// ---- WIND TURBINE/FB_WatsAppResponse.TcPOU
FUNCTION_BLOCK FB_WatsAppResponse
VAR_INPUT
	bSend             : BOOL;
END_VAR
VAR_OUTPUT
	wind_speed		  : Lreal;
	bBusy             : BOOL;
    bError            : BOOL;
END_VAR
VAR
	fbRequest         : FB_IotHttpRequest;
    fbJson            : FB_JsonDomParser;
    nState            : UDINT;
    RisingEdge        : R_TRIG;

    bGetContentResult : BOOL;
    sContent          : STRING(511);

    bGetJsonResult    : BOOL;
    jsonDoc           : SJsonValue;
    jsonVal           : SJsonValue;
	jsonWind           : SJsonValue;

    nReqCount         : UDINT;
    nResCount         : UDINT;
    nValidResCount    : UDINT;
    nErrCount         : UDINT;
	bHasMember		  : BOOL;
	bHasMember2		  : BOOL;
END_VAR
VAR_IN_OUT
	 fbClient          : FB_IotHttpClient;
END_VAR

RisingEdge(CLK:= bSend);
CASE nState OF
0:
    IF RisingEdge.Q THEN
        IF fbRequest.SendRequest(sUri:= '/cebc385e-7c19-40b8-aaac-81ec04618ab7',
                                 fbClient:= fbClient, 
                                 eRequestType:= ETcIotHttpRequestType.HTTP_POST, 0, 0, 0) THEN
            nState:= 1;
            nReqCount:= nReqCount+1;
            bBusy:= TRUE;
            bError:= FALSE;
        END_IF
    END_IF
1:
    IF NOT fbRequest.bBusy THEN
        bError:= TRUE;
        IF NOT fbRequest.bError THEN
            bGetContentResult:= fbRequest.GetContent(pContent:= ADR(sContent), 
                                                     nContentSize:= SIZEOF(sContent), 
                                                     bSetNullTermination:= TRUE);
            IF fbRequest.nStatusCode >= 200 AND fbRequest.nStatusCode < 300 THEN
                bGetJsonResult:= FALSE;
                jsonDoc:= fbRequest.GetJsonDomContent(fbJson);
//                IF jsonDoc <> 0 THEN
//                    bHasMember := fbJson.HasMember(jsonDoc, 'current');
//					IF (bHasMember) THEN
//						bHasMember := FALSE;
//						jsonVal := fbJson.FindMember(jsonDoc, 'current');
//					END_IF
					
//					bHasMember2 := fbJson.HasMember(jsonVal, 'wind_mph');
//					IF (bHasMember2) THEN
//						bHasMember2 := FALSE;
//						jsonWind := fbJson.FindMember(jsonVal, 'wind_mph');
//						wind_speed := fbJson.GetDouble(jsonWind);
//						WindSpeed := fbJson.GetDouble(jsonWind);
//					END_IF
					
//                    nValidResCount:= nValidResCount+1;
//                    bError:= FALSE;
//                END_IF
                nResCount:= nResCount+1;
            END_IF
        END_IF
        nState:= 0;
        bBusy:= FALSE;
        IF bError THEN
            nErrCount:= nErrCount+1;
        END_IF
    END_IF
END_CASE

END_FUNCTION_BLOCK

// ---- BLINDS/BackgroundComms.TcPOU
PROGRAM BackgroundComms
VAR

	HubTXBuffer								:		ARRAY [0..2] OF ComBuffer;
	HubRXBuffer								:		ARRAY [0..2] OF ComBuffer;
                                			        
	HubCommIn AT %I*						:		ARRAY [0..2] OF KL6inData22B;
	HubCommOut AT %Q*						:		ARRAY [0..2] OF KL6outData22B;
                                			        
	HubSerialLineControl					:		ARRAY [0..2] OF SerialLineControl;
                                			        
	i										:		INT;
                                			
	BlindCommandTable 						:		ARRAY [0..2] OF StructBlindControl := [(JogTimeInt:=3000)];
	                            			
	OfficeBlindSellection					:		ARRAY [0..2] OF BOOL;
	                            			
	KitchenBlindSelection					:		BOOL;
	                            			
	BoardroomBlindSellection				:		ARRAY [0..1] OF BOOL;
                                			
	StaffRoomTempDownButton					:		BOOL;
	StaffRoomTempUpButton					:		BOOL;
	StaffRoomTempDownButtonFlag				:		BOOL;
	StaffRoomTempUpButtonFlag				:		BOOL;
	ResetFlagTime 							: 		TON;
                                			
	BlindSelection							:		Selection;
                                			
	UseStaffRoomVisu 						: 		BOOL;
                                			
	Up										:		BOOL;
	Down									:		BOOL;
                                			
	rtBlindsBoardRoomUp						:		R_TRIG;
	rtBlindsBoardRoomDown					:		R_TRIG;
	rtBlindsBoardRoomStop					:		R_TRIG;
	                            			
	rtBlindsOfficeUp						:		R_TRIG;

	(*Office Blinds Triggers *)
	rtBlindsOfficeAreaWall1_3				:		R_TRIG;
	rtBlindsOfficeAreaWall1_3_10_13			:		R_TRIG;
	rtBlindsOfficeAreaWall1_9				:		R_TRIG;
	rtBlindsOfficeAreaWall4_9				:		R_TRIG;
	rtBlindsOfficeAreaWall4_13				:		R_TRIG;
	rtBlindsOfficeAreaWall10_13				:		R_TRIG;
	rtBlindsOfficeAreaWallAll				:		R_TRIG;
	rtBlindsOfficeAreaWallAllFalse			:		R_TRIG;
	
	(*Kitchen Blinds Triggers *)
	rtBlindsKitchenAreaWallAll				:		R_TRIG;
	rtBlindsKitchenAreaWallAllFalse				:		R_TRIG;
	
	(*Boardroom Blinds Triggers *)
	rtBlindsBoardroomAreaWall1_7			:		R_TRIG;
	rtBlindsBoardroomAreaWall8_16			:		R_TRIG;
	rtBlindsBoardroomAreaWallAll			:		R_TRIG;
	rtBlindsBoardroomAreaWallAllFalse		:		R_TRIG;
	
	rtBlindsOfficeAreaWallStop				:		R_TRIG;


	xBlindsOfficeAreaWall1_3Flag			:		BOOL;
	xBlindsOfficeAreaWall4_9Flag			:		BOOL;
	xBlindsOfficeAreaWall10_13Flag			:		BOOL;

	rtBlindsBoardRoomCP67Up					:		R_TRIG;
	rtBlindsBoardRoomCP67Down				:		R_TRIG;
	rtBlindsBoardRoomCP67Stop				:		R_TRIG;


	rtBoardRoom_PrivacyMode					:		R_TRIG;
	rtBoardRoom_SceneryMode					:		R_TRIG;
	rtBoardRoom_ProjectorMode				:		R_TRIG;
	rtBoardRoom_MeetingMode					:		R_TRIG;
                                    		        
	rtDeskArea_PrivacyMode					:		R_TRIG;
	rtDeskArea_SceneryMode					:		R_TRIG;
	rtDeskArea_NightMode					:		R_TRIG;
	rtDeskArea_MorningMode					:		R_TRIG;
                                        	        
	rtKitchenArea_PrivacyMode				:		R_TRIG;
	rtKitchenArea_SceneryMode				:		R_TRIG;
	rtKitchenArea_NightMode					:		R_TRIG;
	rtKitchenArea_MorningMode				:		R_TRIG;
                                        	        
	rtEntireBuilding_CleaningMode			:		R_TRIG;


END_VAR


VAR CONSTANT

	HubCount								:		INT := 2; (* Hub count starts at 0, setting 2 = 3 hubs *)

END_VAR

(* Serial line control for Office Area *)
HubSerialLineControl[0](
	Mode:= SERIALLINEMODE_KL6_22B_STANDARD ,
	pComIn:= ADR( HubCommIn[0]),
	pComOut:= ADR( HubCommOut[0]),
	SizeComIn:=  SIZEOF(HubCommIn[0]),
	TxBuffer:= HubTXBuffer[0] ,
	RxBuffer:= HubRXBuffer[0] ,
	Error=> ,
	ErrorID=> );

(* Serial line control for Boardroom *)
HubSerialLineControl[1](
	Mode:= SERIALLINEMODE_KL6_22B_STANDARD ,
	pComIn:= ADR( HubCommIn[1]),
	pComOut:= ADR( HubCommOut[1]),
	SizeComIn:=  SIZEOF(HubCommIn[1]),
	TxBuffer:= HubTXBuffer[1] ,
	RxBuffer:= HubRXBuffer[1] ,
	Error=> ,
	ErrorID=> );

(*Serial line control for reception *)
HubSerialLineControl[2](
	Mode:= SERIALLINEMODE_KL6_22B_STANDARD ,
	pComIn:= ADR( HubCommIn[2]),
	pComOut:= ADR( HubCommOut[2]),
	SizeComIn:=  SIZEOF(HubCommIn[2]),
	TxBuffer:= HubTXBuffer[2] ,
	RxBuffer:= HubRXBuffer[2] ,
	Error=> ,
	ErrorID=> );

(* Check trigger for boardRoom blinds*)
rtBlindsBoardRoomDown(CLK:= PassADSBlindInfo[2].0 , Q=> );
IF rtBlindsBoardRoomDown.Q THEN
	SetBoardroomAreaBlindsAll();
	BlindCommandTable[1].xCommandDown := TRUE;
END_IF

rtBlindsBoardRoomUp(CLK:= PassADSBlindInfo[3].0 , Q=> );
IF rtBlindsBoardRoomUp.Q THEN
	SetBoardroomAreaBlindsAll();
	BlindCommandTable[1].xCommandUp := TRUE;
END_IF

(*Desk Area Blinds selection******************************************************************)
(*Select Office Blinds and combitanions*)

rtBlindsOfficeAreaWall1_3(CLK := OfficeBlindSellection[0] AND (NOT OfficeBlindSellection[1]) AND (NOT OfficeBlindSellection[2]));
rtBlindsOfficeAreaWall1_3_10_13(CLK := OfficeBlindSellection[0] AND (NOT OfficeBlindSellection[1]) AND OfficeBlindSellection[2]);
rtBlindsOfficeAreaWall1_9(CLK := OfficeBlindSellection[0] AND OfficeBlindSellection[1] AND (NOT OfficeBlindSellection[2]));
rtBlindsOfficeAreaWallAll(CLK := OfficeBlindSellection[0] AND OfficeBlindSellection[1] AND OfficeBlindSellection[2]);
rtBlindsOfficeAreaWall4_9(CLK := (NOT OfficeBlindSellection[0]) AND OfficeBlindSellection[1] AND (NOT OfficeBlindSellection[2]));
rtBlindsOfficeAreaWall4_13(CLK := (NOT OfficeBlindSellection[0]) AND OfficeBlindSellection[1] AND OfficeBlindSellection[2]);
rtBlindsOfficeAreaWall10_13(CLK := (NOT OfficeBlindSellection[0]) AND (NOT OfficeBlindSellection[1]) AND OfficeBlindSellection[2]);
rtBlindsOfficeAreaWallAllFalse(CLK := (NOT OfficeBlindSellection[0]) AND (NOT OfficeBlindSellection[1]) AND (NOT OfficeBlindSellection[2]));

IF rtBlindsOfficeAreaWall1_3.Q THEN
	SetOfficeAreaBlinds1_3();
END_IF

IF rtBlindsOfficeAreaWall1_3_10_13.Q THEN
	SetOfficeAreaBlinds1_3_10_13();
END_IF

IF rtBlindsOfficeAreaWall1_9.Q THEN
	SetOfficeAreaBlinds1_9();
END_IF

IF rtBlindsOfficeAreaWallAll.Q THEN
	SetOfficeAreaBlindsAll();
END_IF

IF rtBlindsOfficeAreaWall4_9.Q THEN
	SetOfficeAreaBlinds4_9();
END_IF

IF rtBlindsOfficeAreaWall4_13.Q THEN
	SetOfficeAreaBlinds4_13();
END_IF

IF rtBlindsOfficeAreaWall10_13.Q THEN
	SetOfficeAreaBlinds10_13();
END_IF

IF rtBlindsOfficeAreaWallAllFalse.Q THEN
	SetOfficeAreaBlindsAllFalse();
END_IF


(*Kitchen Area Blinds selection******************************************************************)
(*Select Kitchen Blinds for Lond Wall*)

rtBlindsKitchenAreaWallAll(CLK := KitchenBlindSelection);
rtBlindsKitchenAreaWallAllFalse(CLK := NOT KitchenBlindSelection);

IF rtBlindsKitchenAreaWallAll.Q THEN
	SetKitchenAreaBlindsAll();
END_IF

IF rtBlindsKitchenAreaWallAllFalse.Q THEN
	SetKitchenAreaBlindsAllFalse();
END_IF

(*Boardroom Area Blinds selection******************************************************************)
(*Select Boardroom Blinds for Lond Wall*)

rtBlindsBoardroomAreaWall1_7(CLK := BoardroomBlindSellection[1] AND (NOT BoardroomBlindSellection[0]));		
rtBlindsBoardroomAreaWall8_16(CLK := (NOT BoardroomBlindSellection[1]) AND BoardroomBlindSellection[0]);
rtBlindsBoardroomAreaWallAll(CLK := BoardroomBlindSellection[0] AND BoardroomBlindSellection[1]);
rtBlindsBoardroomAreaWallAllFalse(CLK := (NOT BoardroomBlindSellection[0]) AND (NOT BoardroomBlindSellection[1]));

IF rtBlindsBoardroomAreaWall1_7.Q THEN
	SetBoardRoomBlinds1_7();
END_IF

IF rtBlindsBoardroomAreaWall8_16.Q THEN
	SetBoardRoomBlinds8_16();
END_IF

IF rtBlindsBoardroomAreaWallAll.Q THEN
	SetBoardroomAreaBlindsAll();
END_IF

IF rtBlindsBoardroomAreaWallAllFalse.Q THEN
	SetBoardroomAreaBlindsAllFalse();
END_IF

(*Boardroom Blind Modes**************************************************************************)
                                                                                        	
(*Board Room Privacy Mode *)                                                            	
rtBoardRoom_PrivacyMode(CLK:= BoardRoom_PrivacyMode , Q=> );                            	
IF rtBoardRoom_PrivacyMode.Q THEN                                                       	
	SetBoardRoomBlinds1_7();                                                            	
	BlindCommandTable[1].xCommandDown := TRUE;                                          	
	BoardRoom_PrivacyMode	:= FALSE;                                                   	
END_IF                                                                                  	
                                                                                        	
(*Board Room Scenery Mode *)                                                            	
rtBoardRoom_SceneryMode(CLK:= BoardRoom_SceneryMode , Q=> );                            	
IF rtBoardRoom_SceneryMode.Q THEN                                                       	
	SetBoardRoomBlinds8_16();                                                           	
	BlindCommandTable[1].xCommandUp := TRUE;                                            	
	BoardRoom_SceneryMode	:= FALSE;                                                   	
END_IF                                                                                  	
                                                                                        	
(*Board Room Projector Mode *)                                                          	
rtBoardRoom_ProjectorMode(CLK:= BoardRoom_ProjectorMode , Q=> );                        	
IF rtBoardRoom_ProjectorMode.Q THEN                                                     	
	SetBoardroomAreaBlindsAll();                                                        	
	BlindCommandTable[1].xCommandDown := TRUE;                                          	
	BoardRoom_ProjectorMode	:= FALSE;                                                   	
END_IF                                                                                  	
                                                                                        	
(*Meeting Room Mode *)                                                                 	
rtBoardRoom_ProjectorMode(CLK:= BoardRoom_ProjectorMode , Q=> );                        	
IF rtBoardRoom_ProjectorMode.Q THEN                                                     	
	SetBoardRoomBlinds1_7();                                                            	
	BlindCommandTable[1].xCommandDown := TRUE;                                          	
	BoardRoom_ProjectorMode	:= FALSE;                                                   	
END_IF                                                                                  	
                                                                                        	
                                                                                        	
(*Desk Area Blind Modes*****************************************************************	******)
                                                                                        	
(* Desk Area Privacy Mode*)                                                             	
rtDeskArea_PrivacyMode(CLK:= DeskArea_PrivacyMode OR PassADSBlindInfo[8].0  , Q=> );    	
IF rtDeskArea_PrivacyMode.Q THEN                                                        	
	SetOfficeAreaBlinds10_13();                                                         	
	BlindCommandTable[0].xCommandDown := TRUE;                                          	
	DeskArea_PrivacyMode	:= FALSE;                                                   	
END_IF                                                                                  	
                                                                                        	
(* Desk Area Scenery Mode*)                                                             	
rtDeskArea_SceneryMode(CLK:= DeskArea_SceneryMode OR  PassADSBlindInfo[11].0  , Q=> );  	
IF rtDeskArea_SceneryMode.Q THEN                                                        	
	SetOfficeAreaBlinds4_9();                                                           	
	BlindCommandTable[0].xCommandUp := TRUE;                                            	
	DeskArea_SceneryMode	:= FALSE;                                                   	
END_IF                                                                                  	
                                                                                        	
(* Desk Area Night Mode*)                                                               	
rtDeskArea_NightMode(CLK:= DeskArea_NightMode OR  PassADSBlindInfo[9].0 , Q=> );        	
IF rtDeskArea_NightMode.Q THEN                                                          	
	SetOfficeAreaBlinds1_9();                                                           	
	BlindCommandTable[0].xCommandDown := TRUE;                                          	
	DeskArea_NightMode	:= FALSE;                                                       	
END_IF                                                                                  	
                                                                                        	
(* Desk Area Morning Mode*)                                                             	
rtDeskArea_MorningMode(CLK:= DeskArea_MorningMode OR  PassADSBlindInfo[10].0 , Q=> );   	
IF rtDeskArea_MorningMode.Q THEN                                                        	
	SetOfficeAreaBlinds1_3();                                                           	
	BlindCommandTable[0].xCommandDown := TRUE;
	DeskArea_MorningMode	:= FALSE;
END_IF

(*Kitchen Area Blind Modes***********************************************************************)

(* Kitchen Area Privacy Mode*)
rtKitchenArea_PrivacyMode(CLK:= KitchenArea_PrivacyMode , Q=> );
IF rtKitchenArea_PrivacyMode.Q THEN
	SetOfficeAreaBlinds10_13();
	SetBoardRoomBlinds1_7();
	BlindCommandTable[0].xCommandDown := TRUE;
	BlindCommandTable[1].xCommandDown := TRUE;
	KitchenArea_PrivacyMode	:= FALSE;
END_IF








(*Check triggers of enocean switch for office area wall 1
rtBlindsOfficeAreaWall1_3(CLK:= PassADSBlindInfo[8].0 , Q=> );
IF rtBlindsOfficeAreaWall1_3.Q AND xBlindsOfficeAreaWall1_3Flag  THEN
	SetOfficeAreaBlinds1_3();
	BlindCommandTable[0].xCommandDown := TRUE;
	xBlindsOfficeAreaWall1_3Flag := FALSE;
ELSIF  rtBlindsOfficeAreaWall1_3.Q AND NOT xBlindsOfficeAreaWall1_3Flag  THEN
	SetOfficeAreaBlinds1_3();
	BlindCommandTable[0].xCommandUp := TRUE;
	xBlindsOfficeAreaWall1_3Flag := TRUE;
END_IF

(*Check triggers of enocean switch for office area wall 2*)
rtBlindsOfficeAreaWall4_9(CLK:= PassADSBlindInfo[9].0 , Q=> );
IF rtBlindsOfficeAreaWall4_9.Q AND xBlindsOfficeAreaWall4_9Flag  THEN
	SetOfficeAreaBlinds4_9();
	BlindCommandTable[0].xCommandDown := TRUE;
	xBlindsOfficeAreaWall4_9Flag := FALSE;
ELSIF  rtBlindsOfficeAreaWall4_9.Q AND NOT xBlindsOfficeAreaWall4_9Flag  THEN
	SetOfficeAreaBlinds4_9();
	BlindCommandTable[0].xCommandUp := TRUE;
	xBlindsOfficeAreaWall4_9Flag := TRUE;
END_IF

(*Check triggers of enocean switch for office area wall 3*)
rtBlindsOfficeAreaWall10_13(CLK:= PassADSBlindInfo[10].0 , Q=> );
IF rtBlindsOfficeAreaWall10_13.Q AND xBlindsOfficeAreaWall10_13Flag  THEN
	SetOfficeAreaBlinds10_13();
	BlindCommandTable[0].xCommandDown := TRUE;
	xBlindsOfficeAreaWall10_13Flag := FALSE;
ELSIF  rtBlindsOfficeAreaWall10_13.Q AND NOT xBlindsOfficeAreaWall10_13Flag  THEN
	SetOfficeAreaBlinds10_13();
	BlindCommandTable[0].xCommandUp := TRUE;
	xBlindsOfficeAreaWall10_13Flag := TRUE;
END_IF


(*Stop*)
rtBlindsOfficeAreaWallStop(CLK:= PassADSBlindInfo[11].0 , Q=> );
IF rtBlindsOfficeAreaWallStop.Q  THEN
	SetOfficeAreaBlindsAll();
	BlindCommandTable[0].xCommandStop := TRUE;
END_IF*)


(* Blind Control from CP67 inputs received via ADS*)

rtBlindsBoardRoomCP67Up(CLK := BYTE_TO_BOOL(PassADSBlindControlCP67[49]));
IF rtBlindsBoardRoomCP67Up.Q THEN

	BlindCommandTable[1].SelectBlindsBulkCommand[1] :=  BYTE_TO_BOOL(PassADSBlindControlCP67[1]);
	BlindCommandTable[1].SelectBlindsBulkCommand[2] :=  BYTE_TO_BOOL(PassADSBlindControlCP67[2]);
	BlindCommandTable[1].SelectBlindsBulkCommand[3] :=  BYTE_TO_BOOL(PassADSBlindControlCP67[3]);
	BlindCommandTable[1].SelectBlindsBulkCommand[4] :=  BYTE_TO_BOOL(PassADSBlindControlCP67[4]);
	BlindCommandTable[1].SelectBlindsBulkCommand[5] :=  BYTE_TO_BOOL(PassADSBlindControlCP67[5]);
	BlindCommandTable[1].SelectBlindsBulkCommand[6] :=  BYTE_TO_BOOL(PassADSBlindControlCP67[6]);
	BlindCommandTable[1].SelectBlindsBulkCommand[7] :=  BYTE_TO_BOOL(PassADSBlindControlCP67[7]);
	BlindCommandTable[1].SelectBlindsBulkCommand[8] :=  BYTE_TO_BOOL(PassADSBlindControlCP67[8]);
	BlindCommandTable[1].SelectBlindsBulkCommand[9] :=  BYTE_TO_BOOL(PassADSBlindControlCP67[9]);
	BlindCommandTable[1].SelectBlindsBulkCommand[10] :=  BYTE_TO_BOOL(PassADSBlindControlCP67[10]);
	BlindCommandTable[1].SelectBlindsBulkCommand[11] :=  BYTE_TO_BOOL(PassADSBlindControlCP67[11]);
	BlindCommandTable[1].SelectBlindsBulkCommand[12] :=  BYTE_TO_BOOL(PassADSBlindControlCP67[12]);
	BlindCommandTable[1].SelectBlindsBulkCommand[13] :=  BYTE_TO_BOOL(PassADSBlindControlCP67[13]);
	BlindCommandTable[1].SelectBlindsBulkCommand[14] :=  BYTE_TO_BOOL(PassADSBlindControlCP67[14]);
	BlindCommandTable[1].SelectBlindsBulkCommand[15] :=  BYTE_TO_BOOL(PassADSBlindControlCP67[15]);
	BlindCommandTable[1].SelectBlindsBulkCommand[16] :=  BYTE_TO_BOOL(PassADSBlindControlCP67[16]);

	BlindCommandTable[1].xCommandUp := TRUE;

END_IF

rtBlindsBoardRoomCP67Down(CLK := BYTE_TO_BOOL(PassADSBlindControlCP67[50]));
IF rtBlindsBoardRoomCP67Down.Q THEN

	BlindCommandTable[1].SelectBlindsBulkCommand[1] :=  BYTE_TO_BOOL(PassADSBlindControlCP67[1]);
	BlindCommandTable[1].SelectBlindsBulkCommand[2] :=  BYTE_TO_BOOL(PassADSBlindControlCP67[2]);
	BlindCommandTable[1].SelectBlindsBulkCommand[3] :=  BYTE_TO_BOOL(PassADSBlindControlCP67[3]);
	BlindCommandTable[1].SelectBlindsBulkCommand[4] :=  BYTE_TO_BOOL(PassADSBlindControlCP67[4]);
	BlindCommandTable[1].SelectBlindsBulkCommand[5] :=  BYTE_TO_BOOL(PassADSBlindControlCP67[5]);
	BlindCommandTable[1].SelectBlindsBulkCommand[6] :=  BYTE_TO_BOOL(PassADSBlindControlCP67[6]);
	BlindCommandTable[1].SelectBlindsBulkCommand[7] :=  BYTE_TO_BOOL(PassADSBlindControlCP67[7]);
	BlindCommandTable[1].SelectBlindsBulkCommand[8] :=  BYTE_TO_BOOL(PassADSBlindControlCP67[8]);
	BlindCommandTable[1].SelectBlindsBulkCommand[9] :=  BYTE_TO_BOOL(PassADSBlindControlCP67[9]);
	BlindCommandTable[1].SelectBlindsBulkCommand[10] :=  BYTE_TO_BOOL(PassADSBlindControlCP67[10]);
	BlindCommandTable[1].SelectBlindsBulkCommand[11] :=  BYTE_TO_BOOL(PassADSBlindControlCP67[11]);
	BlindCommandTable[1].SelectBlindsBulkCommand[12] :=  BYTE_TO_BOOL(PassADSBlindControlCP67[12]);
	BlindCommandTable[1].SelectBlindsBulkCommand[13] :=  BYTE_TO_BOOL(PassADSBlindControlCP67[13]);
	BlindCommandTable[1].SelectBlindsBulkCommand[14] :=  BYTE_TO_BOOL(PassADSBlindControlCP67[14]);
	BlindCommandTable[1].SelectBlindsBulkCommand[15] :=  BYTE_TO_BOOL(PassADSBlindControlCP67[15]);
	BlindCommandTable[1].SelectBlindsBulkCommand[16] :=  BYTE_TO_BOOL(PassADSBlindControlCP67[16]);


	BlindCommandTable[1].xCommandDown := TRUE;

END_IF

rtBlindsBoardRoomCP67Stop(CLK := BYTE_TO_BOOL(PassADSBlindControlCP67[51]));
IF rtBlindsBoardRoomCP67Stop.Q THEN

	BlindCommandTable[1].SelectBlindsBulkCommand[1] :=  BYTE_TO_BOOL(PassADSBlindControlCP67[1]);
	BlindCommandTable[1].SelectBlindsBulkCommand[2] :=  BYTE_TO_BOOL(PassADSBlindControlCP67[2]);
	BlindCommandTable[1].SelectBlindsBulkCommand[3] :=  BYTE_TO_BOOL(PassADSBlindControlCP67[3]);
	BlindCommandTable[1].SelectBlindsBulkCommand[4] :=  BYTE_TO_BOOL(PassADSBlindControlCP67[4]);
	BlindCommandTable[1].SelectBlindsBulkCommand[5] :=  BYTE_TO_BOOL(PassADSBlindControlCP67[5]);
	BlindCommandTable[1].SelectBlindsBulkCommand[6] :=  BYTE_TO_BOOL(PassADSBlindControlCP67[6]);
	BlindCommandTable[1].SelectBlindsBulkCommand[7] :=  BYTE_TO_BOOL(PassADSBlindControlCP67[7]);
	BlindCommandTable[1].SelectBlindsBulkCommand[8] :=  BYTE_TO_BOOL(PassADSBlindControlCP67[8]);
	BlindCommandTable[1].SelectBlindsBulkCommand[9] :=  BYTE_TO_BOOL(PassADSBlindControlCP67[9]);
	BlindCommandTable[1].SelectBlindsBulkCommand[10] :=  BYTE_TO_BOOL(PassADSBlindControlCP67[10]);
	BlindCommandTable[1].SelectBlindsBulkCommand[11] :=  BYTE_TO_BOOL(PassADSBlindControlCP67[11]);
	BlindCommandTable[1].SelectBlindsBulkCommand[12] :=  BYTE_TO_BOOL(PassADSBlindControlCP67[12]);
	BlindCommandTable[1].SelectBlindsBulkCommand[13] :=  BYTE_TO_BOOL(PassADSBlindControlCP67[13]);
	BlindCommandTable[1].SelectBlindsBulkCommand[14] :=  BYTE_TO_BOOL(PassADSBlindControlCP67[14]);
	BlindCommandTable[1].SelectBlindsBulkCommand[15] :=  BYTE_TO_BOOL(PassADSBlindControlCP67[15]);
	BlindCommandTable[1].SelectBlindsBulkCommand[16] :=  BYTE_TO_BOOL(PassADSBlindControlCP67[16]);



	BlindCommandTable[1].xCommandStop := TRUE;

END_IF

ACTION SetBoardroomAreaBlindsAll:
BlindCommandTable[1].SelectBlindsBulkCommand[1] :=TRUE;
BlindCommandTable[1].SelectBlindsBulkCommand[2] := TRUE;
BlindCommandTable[1].SelectBlindsBulkCommand[3] := TRUE;
BlindCommandTable[1].SelectBlindsBulkCommand[4] := TRUE;
BlindCommandTable[1].SelectBlindsBulkCommand[5] := TRUE;
BlindCommandTable[1].SelectBlindsBulkCommand[6] := TRUE;
BlindCommandTable[1].SelectBlindsBulkCommand[7] := TRUE;
BlindCommandTable[1].SelectBlindsBulkCommand[8] := TRUE;
BlindCommandTable[1].SelectBlindsBulkCommand[9] := TRUE;
BlindCommandTable[1].SelectBlindsBulkCommand[10] := TRUE;
BlindCommandTable[1].SelectBlindsBulkCommand[11] := TRUE;
BlindCommandTable[1].SelectBlindsBulkCommand[12] := TRUE;
BlindCommandTable[1].SelectBlindsBulkCommand[13] := TRUE;
BlindCommandTable[1].SelectBlindsBulkCommand[14] := TRUE;
BlindCommandTable[1].SelectBlindsBulkCommand[15] := TRUE;
BlindCommandTable[1].SelectBlindsBulkCommand[16] := TRUE;
END_ACTION

ACTION SetBoardroomAreaBlindsAllFalse:
BlindCommandTable[1].SelectBlindsBulkCommand[1] := FALSE;
BlindCommandTable[1].SelectBlindsBulkCommand[2] := False;
BlindCommandTable[1].SelectBlindsBulkCommand[3] := False;
BlindCommandTable[1].SelectBlindsBulkCommand[4] := False;
BlindCommandTable[1].SelectBlindsBulkCommand[5] := False;
BlindCommandTable[1].SelectBlindsBulkCommand[6] := False;
BlindCommandTable[1].SelectBlindsBulkCommand[7] := False;
BlindCommandTable[1].SelectBlindsBulkCommand[8] := False;
BlindCommandTable[1].SelectBlindsBulkCommand[9] := False;
BlindCommandTable[1].SelectBlindsBulkCommand[10] := FALSE;
BlindCommandTable[1].SelectBlindsBulkCommand[11] := false;
BlindCommandTable[1].SelectBlindsBulkCommand[12] := false;
BlindCommandTable[1].SelectBlindsBulkCommand[13] := false;
BlindCommandTable[1].SelectBlindsBulkCommand[14] := false;
BlindCommandTable[1].SelectBlindsBulkCommand[15] := false;
BlindCommandTable[1].SelectBlindsBulkCommand[16] := false;
END_ACTION

ACTION SetBoardRoomBlinds1_7:
BlindCommandTable[1].SelectBlindsBulkCommand[1] :=TRUE;
BlindCommandTable[1].SelectBlindsBulkCommand[2] := TRUE;
BlindCommandTable[1].SelectBlindsBulkCommand[3] := TRUE;
BlindCommandTable[1].SelectBlindsBulkCommand[4] := TRUE;
BlindCommandTable[1].SelectBlindsBulkCommand[5] := TRUE;
BlindCommandTable[1].SelectBlindsBulkCommand[6] := TRUE;
BlindCommandTable[1].SelectBlindsBulkCommand[7] := TRUE;
BlindCommandTable[1].SelectBlindsBulkCommand[8] := FALSE;
BlindCommandTable[1].SelectBlindsBulkCommand[9] := FALSE;
BlindCommandTable[1].SelectBlindsBulkCommand[10] := FALSE;
BlindCommandTable[1].SelectBlindsBulkCommand[11] := FALSE;
BlindCommandTable[1].SelectBlindsBulkCommand[12] := FALSE;
BlindCommandTable[1].SelectBlindsBulkCommand[13] := FALSE;
BlindCommandTable[1].SelectBlindsBulkCommand[14] := FALSE;
BlindCommandTable[1].SelectBlindsBulkCommand[15] := FALSE;
BlindCommandTable[1].SelectBlindsBulkCommand[16] := FALSE;
END_ACTION

ACTION SetBoardRoomBlinds8_16:
BlindCommandTable[1].SelectBlindsBulkCommand[1] :=FALSE;
BlindCommandTable[1].SelectBlindsBulkCommand[2] := FALSE;
BlindCommandTable[1].SelectBlindsBulkCommand[3] := FALSE;
BlindCommandTable[1].SelectBlindsBulkCommand[4] := FALSE;
BlindCommandTable[1].SelectBlindsBulkCommand[5] := FALSE;
BlindCommandTable[1].SelectBlindsBulkCommand[6] := FALSE;
BlindCommandTable[1].SelectBlindsBulkCommand[7] := FALSE;
BlindCommandTable[1].SelectBlindsBulkCommand[8] := TRUE;
BlindCommandTable[1].SelectBlindsBulkCommand[9] := TRUE;
BlindCommandTable[1].SelectBlindsBulkCommand[10] := TRUE;
BlindCommandTable[1].SelectBlindsBulkCommand[11] := TRUE;
BlindCommandTable[1].SelectBlindsBulkCommand[12] := TRUE;
BlindCommandTable[1].SelectBlindsBulkCommand[13] := TRUE;
BlindCommandTable[1].SelectBlindsBulkCommand[14] := TRUE;
BlindCommandTable[1].SelectBlindsBulkCommand[15] := TRUE;
BlindCommandTable[1].SelectBlindsBulkCommand[16] := TRUE;
END_ACTION

ACTION SetKitchenAreaBlindsAll:
BlindCommandTable[2].SelectBlindsBulkCommand[1] :=TRUE;
BlindCommandTable[2].SelectBlindsBulkCommand[2] := TRUE;
BlindCommandTable[2].SelectBlindsBulkCommand[3] := TRUE;
BlindCommandTable[2].SelectBlindsBulkCommand[4] := TRUE;
BlindCommandTable[2].SelectBlindsBulkCommand[5] := TRUE;
BlindCommandTable[2].SelectBlindsBulkCommand[6] := TRUE;
BlindCommandTable[2].SelectBlindsBulkCommand[7] := TRUE;
BlindCommandTable[2].SelectBlindsBulkCommand[8] := TRUE;
BlindCommandTable[2].SelectBlindsBulkCommand[9] := TRUE;
BlindCommandTable[2].SelectBlindsBulkCommand[10] := TRUE;
BlindCommandTable[2].SelectBlindsBulkCommand[11] := TRUE;
BlindCommandTable[2].SelectBlindsBulkCommand[12] := TRUE;
BlindCommandTable[2].SelectBlindsBulkCommand[13] := TRUE;
BlindCommandTable[2].SelectBlindsBulkCommand[14] := TRUE;
BlindCommandTable[2].SelectBlindsBulkCommand[15] := TRUE;
BlindCommandTable[2].SelectBlindsBulkCommand[16] := TRUE;
END_ACTION

ACTION SetKitchenAreaBlindsAllFalse:
BlindCommandTable[2].SelectBlindsBulkCommand[1] := FALSE;
BlindCommandTable[2].SelectBlindsBulkCommand[2] := false;
BlindCommandTable[2].SelectBlindsBulkCommand[3] := false;
BlindCommandTable[2].SelectBlindsBulkCommand[4] := false;
BlindCommandTable[2].SelectBlindsBulkCommand[5] := false;
BlindCommandTable[2].SelectBlindsBulkCommand[6] := false;
BlindCommandTable[2].SelectBlindsBulkCommand[7] := false;
BlindCommandTable[2].SelectBlindsBulkCommand[8] := false;
BlindCommandTable[2].SelectBlindsBulkCommand[9] := false;
BlindCommandTable[2].SelectBlindsBulkCommand[10] := FALSE;
BlindCommandTable[2].SelectBlindsBulkCommand[11] := false;
BlindCommandTable[2].SelectBlindsBulkCommand[12] := false;
BlindCommandTable[2].SelectBlindsBulkCommand[13] := false;
BlindCommandTable[2].SelectBlindsBulkCommand[14] := false;
BlindCommandTable[2].SelectBlindsBulkCommand[15] := false;
BlindCommandTable[2].SelectBlindsBulkCommand[16] := false;
END_ACTION

ACTION SetOfficeAreaBlinds1_3:
BlindCommandTable[0].SelectBlindsBulkCommand[1] :=TRUE;
BlindCommandTable[0].SelectBlindsBulkCommand[2] := TRUE;
BlindCommandTable[0].SelectBlindsBulkCommand[3] := TRUE;
BlindCommandTable[0].SelectBlindsBulkCommand[4] := FALSE;
BlindCommandTable[0].SelectBlindsBulkCommand[5] := FALSE;
BlindCommandTable[0].SelectBlindsBulkCommand[6] := FALSE;
BlindCommandTable[0].SelectBlindsBulkCommand[7] := FALSE;
BlindCommandTable[0].SelectBlindsBulkCommand[8] := FALSE;
BlindCommandTable[0].SelectBlindsBulkCommand[9] := FALSE;
BlindCommandTable[0].SelectBlindsBulkCommand[10] := FALSE;
BlindCommandTable[0].SelectBlindsBulkCommand[11] := FALSE;
BlindCommandTable[0].SelectBlindsBulkCommand[12] := FALSE;
BlindCommandTable[0].SelectBlindsBulkCommand[13] := FALSE;
BlindCommandTable[0].SelectBlindsBulkCommand[14] := FALSE;
BlindCommandTable[0].SelectBlindsBulkCommand[15] := FALSE;
BlindCommandTable[0].SelectBlindsBulkCommand[16] := FALSE;
END_ACTION

ACTION SetOfficeAreaBlinds1_3_10_13:
BlindCommandTable[0].SelectBlindsBulkCommand[1] :=TRUE;
BlindCommandTable[0].SelectBlindsBulkCommand[2] := TRUE;
BlindCommandTable[0].SelectBlindsBulkCommand[3] := TRUE;
BlindCommandTable[0].SelectBlindsBulkCommand[4] := FALSE;
BlindCommandTable[0].SelectBlindsBulkCommand[5] := FALSE;
BlindCommandTable[0].SelectBlindsBulkCommand[6] := FALSE;
BlindCommandTable[0].SelectBlindsBulkCommand[7] := FALSE;
BlindCommandTable[0].SelectBlindsBulkCommand[8] := FALSE;
BlindCommandTable[0].SelectBlindsBulkCommand[9] := FALSE;
BlindCommandTable[0].SelectBlindsBulkCommand[10] := TRUE;
BlindCommandTable[0].SelectBlindsBulkCommand[11] := TRUE;
BlindCommandTable[0].SelectBlindsBulkCommand[12] := TRUE;
BlindCommandTable[0].SelectBlindsBulkCommand[13] := TRUE;
BlindCommandTable[0].SelectBlindsBulkCommand[14] := TRUE;
BlindCommandTable[0].SelectBlindsBulkCommand[15] := TRUE;
BlindCommandTable[0].SelectBlindsBulkCommand[16] := TRUE;
END_ACTION

ACTION SetOfficeAreaBlinds1_9:
BlindCommandTable[0].SelectBlindsBulkCommand[1] :=TRUE;
BlindCommandTable[0].SelectBlindsBulkCommand[2] := TRUE;
BlindCommandTable[0].SelectBlindsBulkCommand[3] := TRUE;
BlindCommandTable[0].SelectBlindsBulkCommand[4] := TRUE;
BlindCommandTable[0].SelectBlindsBulkCommand[5] := TRUE;
BlindCommandTable[0].SelectBlindsBulkCommand[6] := TRUE;
BlindCommandTable[0].SelectBlindsBulkCommand[7] := TRUE;
BlindCommandTable[0].SelectBlindsBulkCommand[8] := TRUE;
BlindCommandTable[0].SelectBlindsBulkCommand[9] := TRUE;
BlindCommandTable[0].SelectBlindsBulkCommand[10] := FALSE;
BlindCommandTable[0].SelectBlindsBulkCommand[11] := FALSE;
BlindCommandTable[0].SelectBlindsBulkCommand[12] := FALSE;
BlindCommandTable[0].SelectBlindsBulkCommand[13] := FALSE;
BlindCommandTable[0].SelectBlindsBulkCommand[14] := FALSE;
BlindCommandTable[0].SelectBlindsBulkCommand[15] := FALSE;
BlindCommandTable[0].SelectBlindsBulkCommand[16] := FALSE;
END_ACTION

ACTION SetOfficeAreaBlinds10_13:
BlindCommandTable[0].SelectBlindsBulkCommand[1] :=FALSE;
BlindCommandTable[0].SelectBlindsBulkCommand[2] := FALSE;
BlindCommandTable[0].SelectBlindsBulkCommand[3] := FALSE;
BlindCommandTable[0].SelectBlindsBulkCommand[4] := FALSE;
BlindCommandTable[0].SelectBlindsBulkCommand[5] := FALSE;
BlindCommandTable[0].SelectBlindsBulkCommand[6] := FALSE;
BlindCommandTable[0].SelectBlindsBulkCommand[7] := FALSE;
BlindCommandTable[0].SelectBlindsBulkCommand[8] := FALSE;
BlindCommandTable[0].SelectBlindsBulkCommand[9] := FALSE;
BlindCommandTable[0].SelectBlindsBulkCommand[10] := TRUE;
BlindCommandTable[0].SelectBlindsBulkCommand[11] := TRUE;
BlindCommandTable[0].SelectBlindsBulkCommand[12] := TRUE;
BlindCommandTable[0].SelectBlindsBulkCommand[13] := TRUE;
BlindCommandTable[0].SelectBlindsBulkCommand[14] := TRUE;
BlindCommandTable[0].SelectBlindsBulkCommand[15] := TRUE;
BlindCommandTable[0].SelectBlindsBulkCommand[16] := TRUE;
END_ACTION

ACTION SetOfficeAreaBlinds4_13:
BlindCommandTable[0].SelectBlindsBulkCommand[1] :=FALSE;
BlindCommandTable[0].SelectBlindsBulkCommand[2] := FALSE;
BlindCommandTable[0].SelectBlindsBulkCommand[3] := false;
BlindCommandTable[0].SelectBlindsBulkCommand[4] := TRUE;
BlindCommandTable[0].SelectBlindsBulkCommand[5] := TRUE;
BlindCommandTable[0].SelectBlindsBulkCommand[6] := TRUE;
BlindCommandTable[0].SelectBlindsBulkCommand[7] := TRUE;
BlindCommandTable[0].SelectBlindsBulkCommand[8] := TRUE;
BlindCommandTable[0].SelectBlindsBulkCommand[9] := TRUE;
BlindCommandTable[0].SelectBlindsBulkCommand[10] := TRUE;
BlindCommandTable[0].SelectBlindsBulkCommand[11] := TRUE;
BlindCommandTable[0].SelectBlindsBulkCommand[12] := TRUE;
BlindCommandTable[0].SelectBlindsBulkCommand[13] := TRUE;
BlindCommandTable[0].SelectBlindsBulkCommand[14] := TRUE;
BlindCommandTable[0].SelectBlindsBulkCommand[15] := TRUE;
BlindCommandTable[0].SelectBlindsBulkCommand[16] := TRUE;
END_ACTION

ACTION SetOfficeAreaBlinds4_9:
BlindCommandTable[0].SelectBlindsBulkCommand[1] :=FALSE;
BlindCommandTable[0].SelectBlindsBulkCommand[2] := FALSE;
BlindCommandTable[0].SelectBlindsBulkCommand[3] := FALSE;
BlindCommandTable[0].SelectBlindsBulkCommand[4] := TRUE;
BlindCommandTable[0].SelectBlindsBulkCommand[5] := TRUE;
BlindCommandTable[0].SelectBlindsBulkCommand[6] := TRUE;
BlindCommandTable[0].SelectBlindsBulkCommand[7] := TRUE;
BlindCommandTable[0].SelectBlindsBulkCommand[8] := TRUE;
BlindCommandTable[0].SelectBlindsBulkCommand[9] := TRUE;
BlindCommandTable[0].SelectBlindsBulkCommand[10] := FALSE;
BlindCommandTable[0].SelectBlindsBulkCommand[11] := FALSE;
BlindCommandTable[0].SelectBlindsBulkCommand[12] := FALSE;
BlindCommandTable[0].SelectBlindsBulkCommand[13] := FALSE;
BlindCommandTable[0].SelectBlindsBulkCommand[14] := FALSE;
BlindCommandTable[0].SelectBlindsBulkCommand[15] := FALSE;
BlindCommandTable[0].SelectBlindsBulkCommand[16] := FALSE;
END_ACTION

ACTION SetOfficeAreaBlindsAll:
BlindCommandTable[0].SelectBlindsBulkCommand[1] :=TRUE;
BlindCommandTable[0].SelectBlindsBulkCommand[2] := TRUE;
BlindCommandTable[0].SelectBlindsBulkCommand[3] := TRUE;
BlindCommandTable[0].SelectBlindsBulkCommand[4] := TRUE;
BlindCommandTable[0].SelectBlindsBulkCommand[5] := TRUE;
BlindCommandTable[0].SelectBlindsBulkCommand[6] := TRUE;
BlindCommandTable[0].SelectBlindsBulkCommand[7] := TRUE;
BlindCommandTable[0].SelectBlindsBulkCommand[8] := TRUE;
BlindCommandTable[0].SelectBlindsBulkCommand[9] := TRUE;
BlindCommandTable[0].SelectBlindsBulkCommand[10] := TRUE;
BlindCommandTable[0].SelectBlindsBulkCommand[11] := TRUE;
BlindCommandTable[0].SelectBlindsBulkCommand[12] := TRUE;
BlindCommandTable[0].SelectBlindsBulkCommand[13] := TRUE;
BlindCommandTable[0].SelectBlindsBulkCommand[14] := TRUE;
BlindCommandTable[0].SelectBlindsBulkCommand[15] := TRUE;
BlindCommandTable[0].SelectBlindsBulkCommand[16] := TRUE;
END_ACTION

ACTION SetOfficeAreaBlindsAllFalse:
BlindCommandTable[0].SelectBlindsBulkCommand[1] :=FALSE;
BlindCommandTable[0].SelectBlindsBulkCommand[2] := FALSE;
BlindCommandTable[0].SelectBlindsBulkCommand[3] := false;
BlindCommandTable[0].SelectBlindsBulkCommand[4] := FALSE;
BlindCommandTable[0].SelectBlindsBulkCommand[5] := FALSE;
BlindCommandTable[0].SelectBlindsBulkCommand[6] := FALSE;
BlindCommandTable[0].SelectBlindsBulkCommand[7] := FALSE;
BlindCommandTable[0].SelectBlindsBulkCommand[8] := FALSE;
BlindCommandTable[0].SelectBlindsBulkCommand[9] := FALSE;
BlindCommandTable[0].SelectBlindsBulkCommand[10] := FALSE;
BlindCommandTable[0].SelectBlindsBulkCommand[11] := FALSE;
BlindCommandTable[0].SelectBlindsBulkCommand[12] := FALSE;
BlindCommandTable[0].SelectBlindsBulkCommand[13] := FALSE;
BlindCommandTable[0].SelectBlindsBulkCommand[14] := FALSE;
BlindCommandTable[0].SelectBlindsBulkCommand[15] := FALSE;
BlindCommandTable[0].SelectBlindsBulkCommand[16] := FALSE;
END_ACTION

END_PROGRAM

// ---- BLINDS/ADSReadCX9020.TcPOU
PROGRAM ADSReadCX9020
VAR

	UpdateBlindData:ADSREADEX;
	UpdateBlindDataCP67:ADSREADEX;
	UpdateInterval:BYTE;

END_VAR

(* Collects enocean switches from CX9020 SERVER  and CP67 BOARD ROOM*)


UpdateInterval := UpdateInterval + 1;

UpdateBlindData(
	NETID:= '5.129.86.232.1.1',
	PORT:= 851 ,
	IDXGRP:=16#F020,//16#4020 ,
	IDXOFFS:= 16#1F400,//0,
	LEN:= 4,//40,
	DESTADDR:= ADR(PassADSBlindInfo),
	READ:= UpdateInterval.0,
	TMOUT:= t#5s,
	BUSY=> ,
	ERR=> ,
	ERRID=> ,
	COUNT_R=> );



UpdateBlindDataCP67(
	NETID:= '192.168.3.8.1.1',
	PORT:= 851 ,
	IDXGRP:=16#4020 ,
	IDXOFFS:= 40,
	LEN:= 57,
	DESTADDR:= ADR(PassADSBlindControlCP67),
	READ:= UpdateInterval.0,
	TMOUT:= t#5s,
	BUSY=> ,
	ERR=> ,
	ERRID=> ,
	COUNT_R=> );

END_PROGRAM

// ---- ENOCEAN/EnOcean.TcPOU
PROGRAM EnOcean
VAR
	KL6581								:		FB_KL6581;
	
	KL6021FB							:		FB_EnOceanReceive;
	
	EnoceanData							:		ST_EnOceanReceivedData;
	STEnOceanInData		AT %I*			:		ST_EnOceanInData;
	STEnOceanOutData	AT %Q* 			:		ST_EnOceanOutData;
	
	//EnOcean Socket FBs
	fbXplanarScreenPower				:		FB_Send_RPS_Switch; //KL6581 Send Enocen Signals
	
	OpenTennisHMI						:		TON :=(PT := T#2S);;
	TennisHMIOpened						: 		BOOL;	
	
	TEST : ARRAY [0..3] OF BYTE;
	
	i: INT;
	
	AllWindowsClosed				:	bool;
	
	ctudCountWindows				:	ARRAY [0..5] OF CTUD;
	numberOfWindowsOpenTemp			:	ARRAY [0..5] OF WORD;
	totalNumberOfWindowsOpen		:	WORD;
	
	
END_VAR

//FB_KL6581 - Control EnOcean Terminal for transmitting 
KL6581(bInit:=TRUE, nIdx := , stKL6581_in:=stKL6581InData, stKL6581_out:= stKL6581OutData, str_KL6581=> EnOceanComms );
//FB_EnOceanReceive - Control EnOcean Receiver KL6021
KL6021FB(bEnable:= TRUE, stEnOceanReceivedData=> EnoceanData, stEnOceanInData:= STEnOceanInData, stEnOceanOutData:= STEnOceanOutData);	


// Collect all switch data
FOR i := 0 TO 3 DO
	FBEnOceanPTM200[i](
		bEnable:= TRUE, 
		bSwitches =>  ,
		nTransmitterId:= EnoceanTransmitterID[i], 
		stEnOceanReceivedData:= EnoceanData);
END_FOR

FOR i := 0 TO 5 DO	
	FBEnOceanSTM250[i](
		bEnable:= TRUE, 
		nTransmitterId:=EnoceanTransmitterIDWindows[i] , 
		stEnOceanReceivedData:= EnoceanData, 
		bState=> );
END_FOR


//Switches
PTM200StrippedTables[0].Signal := FBEnOceanPTM200[0].bSwitches[0]; // Board Room Bottom Right Off
PTM200StrippedTables[1].Signal := FBEnOceanPTM200[0].bSwitches[1]; // Board Room Bottm Left Off 
PTM200StrippedTables[2].Signal := FBEnOceanPTM200[0].bSwitches[2]; // Board Room Top Right On
PTM200StrippedTables[3].Signal := FBEnOceanPTM200[0].bSwitches[3]; // Board Room Top Left On 
PTM200StrippedTables[4].Signal := FBEnOceanPTM200[1].bSwitches[0]; // Staff Room Bottom Right Off
PTM200StrippedTables[5].Signal := FBEnOceanPTM200[1].bSwitches[1]; // Staff Room Bottom Left Off
PTM200StrippedTables[6].Signal := FBEnOceanPTM200[1].bSwitches[2]; // Staff Room Top Right On
PTM200StrippedTables[7].Signal := FBEnOceanPTM200[1].bSwitches[3]; // Staff Room Top Left On
PTM200StrippedTables[8].Signal := FBEnOceanPTM200[2].bSwitches[0]; //Floating Switch 
PTM200StrippedTables[9].Signal := FBEnOceanPTM200[2].bSwitches[1]; //Floating Switch 
PTM200StrippedTables[10].Signal := FBEnOceanPTM200[2].bSwitches[2]; //Floating Switch 
PTM200StrippedTables[11].Signal := FBEnOceanPTM200[2].bSwitches[3]; //Floating Switch 
PTM200StrippedTables[12].Signal := FBEnOceanPTM200[3].bSwitches[0]; //Tennis Table Left Bottom 
PTM200StrippedTables[13].Signal := FBEnOceanPTM200[3].bSwitches[1]; //Tennis Table Right Bottom  
PTM200StrippedTables[14].Signal := FBEnOceanPTM200[3].bSwitches[2]; //Tennis Table Left Top  
PTM200StrippedTables[15].Signal := FBEnOceanPTM200[3].bSwitches[3]; //Tennis Table Right Top  


//Window States
PTM250WindowSensor[0] := FBEnOceanSTM250[0].bState;
PTM250WindowSensor[1] := FBEnOceanSTM250[1].bState;
PTM250WindowSensor[2] := FBEnOceanSTM250[2].bState; //Window nearest big tele
PTM250WindowSensor[3] := FBEnOceanSTM250[3].bState; //Window nearest coffee machine
PTM250WindowSensor[4] := FBEnOceanSTM250[4].bState; //Window behind Alan's desk
PTM250WindowSensor[5] := FBEnOceanSTM250[5].bState; //Window next to big whiteboard

AllWindowsClosed := PTM250WindowSensor[0] AND PTM250WindowSensor[1] AND PTM250WindowSensor[2] AND PTM250WindowSensor[3] AND PTM250WindowSensor[4] AND PTM250WindowSensor[5];

//Count Open Windows for Dashboard Display
ctudCountWindows[0](
	CU:= NOT PTM250WindowSensor[0], 
	CD:= PTM250WindowSensor[0], 
	PV:= 20, 
	CV=> numberOfWindowsOpenTemp[0]);
	
ctudCountWindows[1](
	CU:= NOT PTM250WindowSensor[1], 
	CD:= PTM250WindowSensor[1], 
	PV:= 20, 
	CV=> numberOfWindowsOpenTemp[1]);
	
ctudCountWindows[2](
	CU:= NOT PTM250WindowSensor[2], 
	CD:= PTM250WindowSensor[2], 
	PV:= 20, 
	CV=> numberOfWindowsOpenTemp[2]);	
	
ctudCountWindows[3](
	CU:= NOT PTM250WindowSensor[3], 
	CD:= PTM250WindowSensor[3], 
	PV:= 20, 
	CV=> numberOfWindowsOpenTemp[3]);

ctudCountWindows[4](
	CU:= NOT PTM250WindowSensor[4], 
	CD:= PTM250WindowSensor[4], 
	PV:= 20, 
	CV=> numberOfWindowsOpenTemp[4]);

ctudCountWindows[5](
	CU:= NOT PTM250WindowSensor[5], 
	CD:= PTM250WindowSensor[5], 
	PV:= 20, 
	CV=> numberOfWindowsOpenTemp[5]);
	
totalNumberOfWindowsOpen := (numberOfWindowsOpenTemp[0] + 
								numberOfWindowsOpenTemp[1] + 
								numberOfWindowsOpenTemp[2] + 
								numberOfWindowsOpenTemp[3] + 
								numberOfWindowsOpenTemp[4] +
								numberOfWindowsOpenTemp[5]);
	
//Collect Switch Data to be collected by CX8090 via ADS READ
(*BlindCommandTable[0] := BOOL_TO_UINT(FBEnOceanPTM200[0].bSwitches[0]); 
BlindCommandTable[1] := BOOL_TO_UINT(FBEnOceanPTM200[0].bSwitches[1]); 
BlindCommandTable[2] := BOOL_TO_UINT(FBEnOceanPTM200[0].bSwitches[2]); 
BlindCommandTable[3] := BOOL_TO_UINT(FBEnOceanPTM200[0].bSwitches[3]);  
BlindCommandTable[4] := BOOL_TO_UINT(FBEnOceanPTM200[1].bSwitches[0]); 
BlindCommandTable[5] := BOOL_TO_UINT(FBEnOceanPTM200[1].bSwitches[1]);  
BlindCommandTable[6] := BOOL_TO_UINT(FBEnOceanPTM200[1].bSwitches[2]); 
BlindCommandTable[7] := BOOL_TO_UINT(FBEnOceanPTM200[1].bSwitches[3]); 
BlindCommandTable[8] := BOOL_TO_UINT(FBEnOceanPTM200[2].bSwitches[0]); 
BlindCommandTable[9] := BOOL_TO_UINT(FBEnOceanPTM200[2].bSwitches[1]); 
BlindCommandTable[10] := BOOL_TO_UINT(FBEnOceanPTM200[2].bSwitches[2]); 
BlindCommandTable[11] := BOOL_TO_UINT(FBEnOceanPTM200[2].bSwitches[3]);  	*)

//Transmit KL6581

//Screen control test ///////////////////////////////////////////////////////////////////////////////////////
//not used for screen anymore - used for display cabinet light
fbXplanarScreenPower(
	bStart:= , 
	by_Node:= 1, 
	bData:= , 
	nRockerID:= 0, 
	nEnOceanID:= 22, 
	str_KL6581:= KL6581.str_KL6581, 
	bBusy=> , 
	bError=> , 
	iErrorID=> );
	
	IF NOT fbXplanarScreenPower.bBusy AND fbXplanarScreenPower.bStart THEN
		fbXplanarScreenPower.bStart := FALSE;
	END_IF

IF xXplanarScreenPowerOn THEN //not used for screen anymore - used for display cabinet light
	fbXplanarScreenPower.bStart := TRUE;
	fbXplanarScreenPower.bData := TRUE;
	xXplanarScreenPowerOn := FALSE;
END_IF

IF xXplanarScreenPowerOff THEN //not used for screen anymore - used for display cabinet light
	fbXplanarScreenPower.bStart := TRUE;
	fbXplanarScreenPower.bData := FALSE;
	xXplanarScreenPowerOff := FALSE;
END_IF


///////////////////////////////////////////////////////////////////////////////////////////////////////////	
TableTennisSwitchHandling();

ACTION TableTennisSwitchHandling:
IF PTM200StrippedTables[12].Signal THEN  // hold in to turn off all before going home
	
	OpenTennisHMI.IN := TRUE;		
	IF OpenTennisHMI.Q THEN
		OpenTennisHMI.IN := FALSE;	
		TennisHMIOpened := TRUE;
	END_IF	
				
END_IF
END_ACTION

END_PROGRAM

// ---- POWER MONITORING/PrgMqttCom_PM_Subscriber.TcPOU
PROGRAM PrgMqttCom_PM_Subscriber
VAR
	fbMqttClient : FB_IotMqttClient;
	bSetParameter : BOOL := TRUE;
	bConnect : BOOL := TRUE;
	
	(* received message *)	
	bSubscribedActivePower : BOOL;
	sTopicActivePower : STRING(255) := 'Active_Power';
	{attribute 'TcEncoding':='UTF-8'}
	sPayloadActivePower : STRING(255);
	
	bSubscribedCurrent : BOOL;
	sTopicCurrent : STRING(255) := 'Current';
	{attribute 'TcEncoding':='UTF-8'}
	sPayloadCurrent : STRING(255);

	bSubscribedVoltage : BOOL;
	sTopicVoltage : STRING(255) := 'Voltage';
	{attribute 'TcEncoding':='UTF-8'}
	sPayloadVoltage : STRING(255);

	bSubscribedApparentPower : BOOL;	
	sTopicApparentPower	: STRING(255) := 'Apparent_Power';
	{attribute 'TcEncoding':='UTF-8'}
	sPayloadApparentPower : STRING(255);

	bSubscribedReactivePower : BOOL;	
	sTopicReactivePower	: STRING(255) := 'Reactive_Power';
	{attribute 'TcEncoding':='UTF-8'}
	sPayloadReactivePower : STRING(255);

	bSubscribedPositiveEnergy : BOOL;	
	sTopicPositiveEnergy	: STRING(255) := 'Positive_Energy';
	{attribute 'TcEncoding':='UTF-8'}
	sPayloadPositiveEnergy : STRING(255);

	bSubscribedCosPhi : BOOL;
	sTopicCosPhi	: STRING(255) := 'cosPhi';
	{attribute 'TcEncoding':='UTF-8'}
	sPayloadCosPhi : STRING(255);	

	bSubscribedFrequency : BOOL;	
	sTopicFrequency	: STRING(255) := 'Frequency';
	{attribute 'TcEncoding':='UTF-8'}
	sPayloadFrequency : STRING(255);
	
	bSubscribedNegativeEnergy : BOOL;
	sTopicNegativeEnergy	: STRING(255) := 'Negative_Energy';
	{attribute 'TcEncoding':='UTF-8'}
	sPayloadNegativeEnergy : STRING(255);		
	
	powerData				:	ST_EL3403_Data;
	scaledPowerData			:	ST_EL3403_Data;
		
	fbMessageQueue : FB_IotMqttMessageQueue;
	fbMessage : FB_IotMqttMessage;
	
	hrErrorOccurred : HRESULT; // contains the latest occurred error
END_VAR

IF bSetParameter THEN
	bSetParameter := FALSE;
	fbMqttClient.sHostName:= '10.199.143.2';
	fbMqttClient.nHostPort:= 1883;
	fbMqttClient.sClientId:= 'CX2040_Power_Monitoring'; 
	fbMqttClient.sTopicPrefix:= ''; 
	fbMqttClient.nKeepAlive:= 60; 
	fbMqttClient.ipMessageQueue := fbMessageQueue;
END_IF

fbMqttClient.Execute(bConnect);
IF fbMqttClient.bError THEN
	// add your error logging here
	hrErrorOccurred := fbMqttClient.hrErrorCode;
END_IF

IF fbMessageQueue.nQueuedMessages > 0 THEN
	IF fbMessageQueue.Dequeue(fbMessage:=fbMessage) THEN
		IF fbMessage.CompareTopic(sTopic := sTopicVoltage) THEN
			fbMessage.GetPayload(pPayload:=ADR(sPayloadVoltage), nPayloadSize:=SIZEOF(sPayloadVoltage), bSetNullTermination:=FALSE);
        	powerData.voltage := STRING_TO_REAL(sPayloadVoltage);
			
		ELSIF fbMessage.CompareTopic(sTopic:=sTopicCurrent) THEN
            fbMessage.GetPayload(pPayload:=ADR(sPayloadCurrent), nPayloadSize:=SIZEOF(sPayloadCurrent), bSetNullTermination:=FALSE);
        	powerData.current := STRING_TO_REAL(sPayloadCurrent);
			
		ELSIF fbMessage.CompareTopic(sTopic:=sTopicActivePower) THEN
            fbMessage.GetPayload(pPayload:=ADR(sPayloadActivePower), nPayloadSize:=SIZEOF(sPayloadActivePower), bSetNullTermination:=FALSE);
        	powerData.activePower := STRING_TO_REAL(sPayloadActivePower);

		ELSIF fbMessage.CompareTopic(sTopic:=sTopicReactivePower) THEN
            fbMessage.GetPayload(pPayload:=ADR(sPayloadReactivePower), nPayloadSize:=SIZEOF(sPayloadReactivePower), bSetNullTermination:=FALSE);
        	powerData.reactivePower := STRING_TO_REAL(sPayloadReactivePower);
						
		ELSIF fbMessage.CompareTopic(sTopic:=sTopicApparentPower) THEN
            fbMessage.GetPayload(pPayload:=ADR(sPayloadApparentPower), nPayloadSize:=SIZEOF(sPayloadApparentPower), bSetNullTermination:=FALSE);
        	powerData.apparentPower := STRING_TO_REAL(sPayloadApparentPower);
			
		ELSIF fbMessage.CompareTopic(sTopic:=sTopicFrequency) THEN
            fbMessage.GetPayload(pPayload:=ADR(sPayloadFrequency), nPayloadSize:=SIZEOF(sPayloadFrequency), bSetNullTermination:=FALSE);
        	powerData.frequency := STRING_TO_REAL(sPayloadFrequency);

		ELSIF fbMessage.CompareTopic(sTopic:=sTopicPositiveEnergy) THEN
            fbMessage.GetPayload(pPayload:=ADR(sPayloadPositiveEnergy), nPayloadSize:=SIZEOF(sPayloadPositiveEnergy), bSetNullTermination:=FALSE);
        	powerData.positiveEnergy := STRING_TO_REAL(sPayloadPositiveEnergy);
			
		ELSIF fbMessage.CompareTopic(sTopic:=sTopicNegativeEnergy) THEN
            fbMessage.GetPayload(pPayload:=ADR(sPayloadNegativeEnergy), nPayloadSize:=SIZEOF(sPayloadNegativeEnergy), bSetNullTermination:=FALSE);
        	powerData.negativeEnergy := STRING_TO_REAL(sPayloadNegativeEnergy);

		ELSIF fbMessage.CompareTopic(sTopic:=sTopicCosPhi) THEN
            fbMessage.GetPayload(pPayload:=ADR(sPayloadCosPhi), nPayloadSize:=SIZEOF(sPayloadCosPhi), bSetNullTermination:=FALSE);
        	powerData.cosPhi := STRING_TO_REAL(sPayloadCosPhi);								
		END_IF
	END_IF
END_IF

IF fbMqttClient.bConnected THEN
	IF NOT bSubscribedVoltage THEN
		bSubscribedVoltage := fbMqttClient.Subscribe(sTopic:=sTopicVoltage, eQoS:=TcIotMqttQos.AtMostOnceDelivery);
		IF fbMqttClient.bError THEN
			// add your error logging here
			hrErrorOccurred := fbMqttClient.hrErrorCode;
		END_IF
	END_IF	

	IF NOT bSubscribedCurrent THEN
		bSubscribedCurrent := fbMqttClient.Subscribe(sTopic:=sTopicCurrent, eQoS:=TcIotMqttQos.AtMostOnceDelivery);
		IF fbMqttClient.bError THEN
			// add your error logging here
			hrErrorOccurred := fbMqttClient.hrErrorCode;
		END_IF
	END_IF
	
	IF NOT bSubscribedActivePower THEN
		bSubscribedActivePower := fbMqttClient.Subscribe(sTopic:=sTopicActivePower, eQoS:=TcIotMqttQos.AtMostOnceDelivery);
		IF fbMqttClient.bError THEN
			// add your error logging here
			hrErrorOccurred := fbMqttClient.hrErrorCode;
		END_IF
	END_IF

	IF NOT bSubscribedApparentPower THEN
		bSubscribedApparentPower := fbMqttClient.Subscribe(sTopic:=sTopicApparentPower, eQoS:=TcIotMqttQos.AtMostOnceDelivery);
		IF fbMqttClient.bError THEN
			// add your error logging here
			hrErrorOccurred := fbMqttClient.hrErrorCode;
		END_IF
	END_IF
	
	IF NOT bSubscribedReactivePower THEN
		bSubscribedApparentPower := fbMqttClient.Subscribe(sTopic:=sTopicReactivePower, eQoS:=TcIotMqttQos.AtMostOnceDelivery);
		IF fbMqttClient.bError THEN
			// add your error logging here
			hrErrorOccurred := fbMqttClient.hrErrorCode;
		END_IF
	END_IF
	
	IF NOT bSubscribedPositiveEnergy THEN
		bSubscribedPositiveEnergy := fbMqttClient.Subscribe(sTopic:=sTopicPositiveEnergy, eQoS:=TcIotMqttQos.AtMostOnceDelivery);
		IF fbMqttClient.bError THEN
			// add your error logging here
			hrErrorOccurred := fbMqttClient.hrErrorCode;
		END_IF
	END_IF
	
	IF NOT bSubscribedCosPhi THEN
		bSubscribedCosPhi := fbMqttClient.Subscribe(sTopic:=sTopicCosPhi, eQoS:=TcIotMqttQos.AtMostOnceDelivery);
		IF fbMqttClient.bError THEN
			// add your error logging here
			hrErrorOccurred := fbMqttClient.hrErrorCode;
		END_IF
	END_IF
	
	IF NOT bSubscribedFrequency THEN
		bSubscribedFrequency := fbMqttClient.Subscribe(sTopic:=sTopicFrequency, eQoS:=TcIotMqttQos.AtMostOnceDelivery);
		IF fbMqttClient.bError THEN
			// add your error logging here
			hrErrorOccurred := fbMqttClient.hrErrorCode;
		END_IF
	END_IF
	
	IF NOT bSubscribedNegativeEnergy THEN
		bSubscribedNegativeEnergy := fbMqttClient.Subscribe(sTopic:=sTopicNegativeEnergy, eQoS:=TcIotMqttQos.AtMostOnceDelivery);
		IF fbMqttClient.bError THEN
			// add your error logging here
			hrErrorOccurred := fbMqttClient.hrErrorCode;
		END_IF
	END_IF
END_IF

PowerScaling();

METHOD PowerScaling : BOOL
VAR_INPUT
END_VAR
//Scaled to A
scaledPowerData.current         := (powerData.current * 0.000001 * 10); 

//Scaled to Vac        
scaledPowerData.voltage         := (powerData.voltage * 0.0001);  

//Scaled to Hz      
scaledPowerData.frequency       := (powerData.frequency * 0.1);    

//Scaled to W
scaledPowerData.activePower     := (powerData.activePower * 0.01);   

//Scaled to W  
scaledPowerData.apparentPower   := (powerData.apparentPower * 0.01); 

//Scaled to VAr  
scaledPowerData.reactivePower   := (powerData.reactivePower * 0.01);  

//Scaled to Wh  
scaledPowerData.positiveEnergy  := ((powerData.positiveEnergy * 0.001)*10);  

//Scaled to WH 
scaledPowerData.negativeEnergy  := (powerData.negativeEnergy * 0.001);  

//Power factor
scaledPowerData.cosPhi			:= (powerData.cosPhi * 0.001);
END_METHOD

END_PROGRAM

// ---- LIGHTS/DALI/Dali.TcPOU
PROGRAM Dali
VAR
	KL6811_Tc2							:			Tc2_DALI.FB_DALIV2Communication;
	KL6811_Tc3							:			Tc3_DALI.FB_KL6811Communication;
	
	
	bAssumeBuildingEmpty			:			BOOL;
	TONGlobalMovementTimer			:			TON;


	CommunalAreaPIR_1:FB_DALIV2IAPIR;
	{attribute 'OPC.UA.DA' := '1'}
	CommunalAreaPIR_1_Occupancy:BOOL;(*~ (OPC:1:available) *)
	{attribute 'OPC.UA.DA' := '1'}
	CommunalAreaPIR_1_LuxLevel:INT;(*~ (OPC:1:available) *)
	{attribute 'OPC.UA.DA' := '1'}
	CommunalAreaPIR_2:FB_DALIV2IAPIR;
	{attribute 'OPC.UA.DA' := '1'}
	CommunalAreaPIR_2_Occupancy:BOOL;(*~ (OPC:1:available) *)
	{attribute 'OPC.UA.DA' := '1'}
	CommunalAreaPIR_2_LuxLevel:INT;(*~ (OPC:1:available) *)
	{attribute 'OPC.UA.DA' := '1'}
	StaffroomPIR_1:FB_DALIV2IAPIR;
	{attribute 'OPC.UA.DA' := '1'}
	StaffroomPIR_1_Occupancy:BOOL;(*~ (OPC:1:available) *)
	{attribute 'OPC.UA.DA' := '1'}
	StaffroomPIR_1_LuxLevel:INT;(*~ (OPC:1:available) *)
	{attribute 'OPC.UA.DA' := '1'}
	StaffroomPIR_2:FB_DALIV2IAPIR;
	{attribute 'OPC.UA.DA' := '1'}
	StaffroomPIR_2_Occupancy:BOOL; (*~ (OPC:1:available) *)
	{attribute 'OPC.UA.DA' := '1'}
	StaffroomPIR_2_LuxLevel:INT;(*~ (OPC:1:available) *)
	{attribute 'OPC.UA.DA' := '1'}
	BoardroomPIR_1:FB_DALIV2IAPIR;
	{attribute 'OPC.UA.DA' := '1'}
	BoardroomPIR_1_Occupancy:BOOL;(*~ (OPC:1:available) *)
	{attribute 'OPC.UA.DA' := '1'}
	BoardroomPIR_1_LuxLevel:INT;(*~ (OPC:1:available) *)
	{attribute 'OPC.UA.DA' := '1'}
	BoardroomPIR_2:FB_DALIV2IAPIR;
	{attribute 'OPC.UA.DA' := '1'}
	BoardroomPIR_2_Occupancy:BOOL;(*~ (OPC:1:available) *)
	{attribute 'OPC.UA.DA' := '1'}
	BoardroomPIR_2_LuxLevel:INT;(*~ (OPC:1:available) *)
	{attribute 'OPC.UA.DA' := '1'}
	CommunalAreaLights:FB_DALIV2DirectArcPowerControl;
	{attribute 'OPC.UA.DA' := '1'}
	CommunalAreaLightsLevel:BYTE;(*~ (OPC:1:available) *)
	{attribute 'OPC.UA.DA' := '1'}
	StaffroomLights:FB_DALIV2DirectArcPowerControl;
	{attribute 'OPC.UA.DA' := '1'}
	StaffroomLightsLevel:BYTE;(*~ (OPC:1:available) *)
	{attribute 'OPC.UA.DA' := '1'}
	BoardroomBackLights:FB_DALIV2DirectArcPowerControl;
	{attribute 'OPC.UA.DA' := '1'}
	BoardroomBackLightsLevel:BYTE;(*~ (OPC:1:available) *)
	{attribute 'OPC.UA.DA' := '1'}
	BoardroomFrontLights:FB_DALIV2DirectArcPowerControl;
	{attribute 'OPC.UA.DA' := '1'}
	BoardroomFrontLightsLevel:BYTE;(*~ (OPC:1:available) *)

	i: BYTE;
END_VAR

KL6811_Tc2(
	bResetMaximumDemandCounter:= ,
	bResetOverflowCounter:= ,
	stDALIInData:=  stDALIInData ,
	stDALIOutData:= stDALIOutData ,
	stCommandBuffer:= stCommandBuffer ,
	arrBufferDemandMeter=> ,
	arrBufferMaximumDemandMeter=> ,
	arrBufferOverflowCounter=> , 
	bLineIsBusy=> ,
	bLineIsInitialized=> );
	
	//stKL6811InData.nData := stDALIInData.nData;
	//stKL6811InData.nStatus :=  stDALIInData.nStatus;
	
	//stKL6811OutData.nCtrl := stDALIOutData.nCtrl;
	//stKL6811OutData.nData := stDALIOutData.nData;
	
KL6811_Tc3(
	bError=> , 
	ipResultMessage=> , 
	bResetMaximumDemandCounter:= , 
	bResetOverflowCounter:= , 
	nOptions:= , 
	bBusy=> , 
	nBufferDemandMeter=> , 
	nBufferMaximumDemandMeter=> , 
	nBufferOverflowCounter=> , 
	bInitialise:= , 
	bDisableInternalPowerSupply:= , 
	bCollisionErrorFC=> , 
	bCollisionErrorBC=> , 
	bPowerSupplyError=> , 
	bInitialising=> , 
	nTerminalDescription=> , 
	nFirmwareVersion=> , 
	stInData:= stKL6811InData, 
	stOutData:= stKL6811OutData);

	// Check Building Occupancy
	TONGlobalMovementTimer(PT := T#3H );
	IF NOT Dali.BoardroomPIR_1_Occupancy AND NOT Dali.BoardroomPIR_2_Occupancy AND NOT Dali.CommunalAreaPIR_1_Occupancy AND NOT Dali.CommunalAreaPIR_2_Occupancy AND NOT Dali.StaffroomPIR_1_Occupancy AND NOT Dali.StaffroomPIR_2_Occupancy THEN
		TONGlobalMovementTimer.IN := TRUE;
	ELSE
		TONGlobalMovementTimer.IN := FALSE;
		bAssumeBuildingEmpty := FALSE;
	END_IF
	
	IF TONGlobalMovementTimer.Q THEN
		bAssumeBuildingEmpty := TRUE;
	END_IF
	


	
// Room Sensors PIR	
BoardroomPIR_1(
	nAddr:=0 ,
	eAddrType:=0 ,
	stCommandBuffer:=stCommandBuffer ,
	bOccupancy=>BoardroomPIR_1_Occupancy ,
	nBrightness=>BoardroomPIR_1_LuxLevel );
	
BoardroomPIR_2(
	nAddr:=1 ,
	eAddrType:=0 ,
	stCommandBuffer:=stCommandBuffer  ,
	bOccupancy=>BoardroomPIR_2_Occupancy ,
	nBrightness=>BoardroomPIR_2_LuxLevel );

CommunalAreaPIR_1(
	nAddr:=2 ,
	eAddrType:=0 ,
	stCommandBuffer:=stCommandBuffer ,
	bOccupancy=>CommunalAreaPIR_1_Occupancy ,
	nBrightness=>CommunalAreaPIR_1_LuxLevel  );
	
CommunalAreaPIR_2(
	nAddr:=3 ,
	eAddrType:=0 ,
	stCommandBuffer:=stCommandBuffer ,
	bOccupancy=>CommunalAreaPIR_2_Occupancy ,
	nBrightness=>CommunalAreaPIR_2_LuxLevel );

StaffroomPIR_1(
	nAddr:=4 ,
	eAddrType:=0 ,
	stCommandBuffer:=stCommandBuffer ,
	bOccupancy=>StaffroomPIR_1_Occupancy ,
	nBrightness=>StaffroomPIR_1_LuxLevel  );
	
StaffroomPIR_2(
	nAddr:=5 ,
	eAddrType:=0 ,
	stCommandBuffer:=stCommandBuffer ,
	bOccupancy=>StaffroomPIR_2_Occupancy ,
	nBrightness=>StaffroomPIR_2_LuxLevel  );
	
	
(*
BoardroomBackLights(
	bStart:= NOT BoardroomBackLights.bBusy ,
	nAddr:=2 ,
	eAddrType:=1 ,
	nArcPowerLevel:=BoardroomBackLightsLevel ,
	stCommandBuffer:=stCommandBuffer  );

BoardroomFrontLights(
	bStart:=NOT BoardroomFrontLights.bBusy,
	nAddr:=3 ,
	eAddrType:=1 ,
	nArcPowerLevel:=BoardroomFrontLightsLevel ,
	stCommandBuffer:=stCommandBuffer  );

CommunalAreaLights(
	bStart:=NOT CommunalAreaLights.bBusy ,
	nAddr:=0 ,
	eAddrType:=1 ,
	nArcPowerLevel:=CommunalAreaLightsLevel ,
	stCommandBuffer:=stCommandBuffer  );

StaffroomLights(
	bStart:=NOT StaffroomLights.bBusy ,
	nAddr:=1 ,
	eAddrType:=1 ,
	nArcPowerLevel:=StaffroomLightsLevel ,
	stCommandBuffer:=stCommandBuffer  );*)

END_PROGRAM

// ---- LIGHTS/DALI/LightControl.TcPOU
PROGRAM LightControl
VAR
	
	//Force Variables
	TurnAllOff								:	BOOL;
	TurnAllOn								:	BOOL;
	Bypass									:	BOOL;
	
	//UPdate light status pulse
	Update									:	INT;	
	
	//Set Min Or Max Levels
	SetMaxLevel								:	FB_DALIV2SetMaxLevel;
	xExecuteSetMax							:	BOOL;
	MaxSetting								:	BYTE := 255;
	SetMinLevel								:	FB_DALIV2SetMinLevel;
	xExecuteSetMin							:	BOOL;
	MinSetting								:	BYTE := 76;	
  	DaliAddrress							:	BYTE;
	                                    	
                                        	
                                        	
	//Group Light OFF control           	
	TurnAllOffGroup0_MiddleRoom				:	FB_DALIV2Off;		
	TurnAllOffGroup1_OfficeDesks			:	FB_DALIV2Off;
	TurnAllOffGroup2_BoardroomBackRow		:	FB_DALIV2Off;
	TurnAllOffGroup3_BoardroomFront2		:	FB_DALIV2Off;
	TurnAllOffGroup4_OfficePassage			:	FB_DALIV2Off;
	TurnAllOffGroup5_SmallBoardRoom			:	FB_DALIV2Off;
	TurnAllOffGroup6_MiddleRoomPassage		:	FB_DALIV2Off;
	TurnAllOffGroup7_TechRoom				:	FB_DALIV2Off;
	TurnAllOffGroup8_ServerRoom				:	FB_DALIV2Off;
	
	
	//Light Control Per Group
	LightControlGroup0_MiddleRoom			:	FB_DALIV2Light;
	LightControlGroup1_OfficeDesks			:	FB_DALIV2Light;
	LightControlGroup2_BoardroomBackRow		:	FB_DALIV2Light;
	LightControlGroup3_BoardroomFront2		:	FB_DALIV2Light;
	LightControlGroup4_OfficePassage		:	FB_DALIV2Light;
	LightControlGroup5_SmallBoardRoom		:	FB_DALIV2Light;
	LightControlGroup6_MiddleRoomPassage	:	FB_DALIV2Light;
	LightControlGroup7_TechRoom				:	FB_DALIV2Light;
	LightControlGroup8_ServerRoom			:	FB_DALIV2Light;
	
	//Recall Max Level			
	RecallMaxLevelGroup0_MiddleRoom			:	FB_DALIV2RecallMaxLevel;
	RecallMaxLevelGroup1_OfficeDesks		:	FB_DALIV2RecallMaxLevel;
	RecallMaxLevelGroup2_BoardroomBackRow	:	FB_DALIV2RecallMaxLevel;
	RecallMaxLevelGroup3_BoardroomFront2	:	FB_DALIV2RecallMaxLevel;
	RecallMaxLevelGroup4_OfficePassage		:	FB_DALIV2RecallMaxLevel;
	RecallMaxLevelGroup5_SmallBoardRoom		:	FB_DALIV2RecallMaxLevel;
	RecallMaxLevelGroup6_MiddleRoomPassage	:	FB_DALIV2RecallMaxLevel;
	RecallMaxLevelGroup7_TechRoom			:	FB_DALIV2RecallMaxLevel;
	RecallMaxLevelGroup8_ServerRoom			:	FB_DALIV2RecallMaxLevel;
	
	//Recall Min Level		
	//Groups	
	RecallMinLevelGroup0_MiddleRoom			:	FB_DALIV2RecallMinLevel;
	RecallMinLevelGroup1_OfficeDesks		:	FB_DALIV2RecallMinLevel;
	RecallMinLevelGroup2_BoardroomBackRow	:	FB_DALIV2RecallMinLevel;
	RecallMinLevelGroup3_BoardroomFront2	:	FB_DALIV2RecallMinLevel;
	RecallMinLevelGroup4_OfficePassage		:	FB_DALIV2RecallMinLevel;
	RecallMinLevelGroup5_SmallBoardRoom		:	FB_DALIV2RecallMinLevel;
	RecallMinLevelGroup6_MiddleRoomPassage	:	FB_DALIV2RecallMinLevel;
	RecallMinLevelGroup7_TechRoom			:	FB_DALIV2RecallMinLevel;
	RecallMinLevelGroup8_ServerRoom			:	FB_DALIV2RecallMinLevel;
	
	//Individual Lamps
	RecallMinLevelCouchLight				:	FB_DALIV2RecallMinLevel;
	RecallStepUPCouchLight					:	FB_DALIV2StepUp;
	
	IgnoreFronttime : ton;
	
	

	nForceLightsOffHour						:	INT := 19;	// Lights will turn off at this time
	nHourOfDay								:	INT;
	bNoOccupancyFlag						:	BOOL;
	trigbAssumeBuildingEmpty				:	R_TRIG;
	i										:	BYTE;
                                        	
	FBDALIV2Dimmer1SwitchStaff				:	FB_DALIV2Dimmer1Switch;
	FBDALIV2Dimmer1SwitchBoarda				:	FB_DALIV2Dimmer1Switch;	
	FBDALIV2Dimmer1SwitchBoardb				:	FB_DALIV2Dimmer1Switch;
	FBDALIV2Dimmer1SwitchBoardc				:	FB_DALIV2Dimmer1Switch;
	FBDALIV2Dimmer1SwitchBoardd				:	FB_DALIV2Dimmer1Switch;
	FBDALIV2Dimmer1SwitchBoarde				:	FB_DALIV2Dimmer1Switch;
	FBDALIV2Dimmer1SwitchBoardf				:	FB_DALIV2Dimmer1Switch;
				                        	
	                                    	
	                                    	
	OfficeDimmValue							:	BYTE := 190;	
	WorkshopDimmValue						:	BYTE := 190;
	                                    	
	FBFade									:	FB_DALIV2Ramp;
	
	FBFadeOffice							:	FB_DALIV2Dimmer1Switch;
	FBFadeWorkshop							:	FB_DALIV2Dimmer1Switch;
		
	bMainEntranceFadeSetFlag				:	BOOL;
	nEndLevelIn								:	BYTE;
	MainEntTimer							:	TON;
	OfficeTimer								:	TON;
	                                    	
	bMainOfficeFadeSetFlag					: 	BOOL;       	
	                                    	
	OfficeLightControl						:	FB_ConstantLightControlEco;
	WorkshopLightControl					:	FB_ConstantLightControlEco;
	OfficePassageLightControl				:	FB_DALIV2Light;
	ServerRoomLightControl					:	FB_DALIV2Light;
	                                    	
	EmergancyLightControlOffice				:	FB_DALIV2RecallMaxLevel;
	EmergancyLightControlBoard				:	FB_DALIV2Light;
	EmergancyLightControlReception			:	FB_DALIV2Light;
	
	ReceptionDoorLightControl				:	FB_DALIV2Light;
	ReceptionPassageLightControl			:	FB_DALIV2Light;
	ReceptionTableKitchLoungeLightControl	:	FB_DALIV2Light;
	
	ReceptionDoorLightControlOnLeave		:	FB_DALIV2Light;
	
	
	SmallBoardRoomLightControl				:	FB_DALIV2Light;
	SmallBoardRoomDimm						:	FB_DALIV2Dimmer1Switch;
	SmallBoardRoomOff						:	FB_DALIV2Off;
	
	
	SmallBoardRoomTime						:	TON;
	SmallBoardRoomTriggerOn					:	BOOL;
	SmallBoardRoomTriggerOff				:	BOOL;
	                                    	
	                                    	
	OfficePassageTime						:	TON;
	OfficePassageTriggerOn					:	BOOL;
	OfficePassageTriggerOff					:	BOOL;	
	                                    	
	WorkshopPassageTime						:	TON;
	WorkshopPassageTriggerOn				:	BOOL;
	WorkshopPassageTriggerOff				:	BOOL;
	                                    	
	DeskAreaTime							:	TON;
	DeskAreaTriggerOn						:	BOOL;
	DeskAreaTriggerOff						:	BOOL;
	                                    	
	OfficeLightLevel						:	UINT;
	WorkshopLightLevel						:	UINT;
	
	BoardRoomTime							:	Ton;
	BoardRoomTriggerOn						:	BOOL;
	BoardRoomTriggerOff						:	BOOL;
	
	
	bLightADS 					AT %MB100	:	BOOL;
	bLightsADSOff 				AT %MB110 	:	BOOL;
	

	ReceptionDoorTriggerOn					:	BOOL;
	ReceptionDoorTriggerOFF					:	BOOL;
	
	ReceptionPassageTriggerOn				:	BOOL;
	ReceptionPassageTriggerOFF				:	BOOL;
	                                		 	
		                            		 	
	                                		 	
	ReceptionDoorTime						:	TON;
	ReceptionPassageTime					:	TON;
	ReceptionTableKitchLoungeTime			:	TON;
	                                		 	
	
	GoHomeHold 								:	TON;
	GoHomeHoldActivated						:	BOOL;
	ClearRoomTimer							:	TON;
	

	
	ResetOthers								:	BOOL;
	ReceptionTableKitchLoungeTriggerOn		:	BOOL;
	ReceptionTableKitchLoungeTriggerOFF		:	BOOL;
	
	OfficeLightLevelSetpoint				:	UINT := 900;
	WorkshopLightLevelSetpoint				:	UINT := 1000;
	
	xBoardRoom_Lights_ProjectorMode			:	BOOL;
	xBoardRoom_Lights_ShowroomMode			:	BOOL;
	rt_BoardRoom_Lights_ProjectorMode		:	R_TRIG;
	rt_BoardRoom_Lights_ShowroomMode		:	R_TRIG;
	
	rt_BoardRoom_Lights_Switch0				:	R_TRIG := (CLK := PTM200StrippedTables[0].Signal);
	rt_BoardRoom_Lights_Switch1				:	R_TRIG := (CLK := PTM200StrippedTables[1].Signal);
	rt_BoardRoom_Lights_Switch2				:	R_TRIG := (CLK := PTM200StrippedTables[2].Signal);
	rt_BoardRoom_Lights_Switch3				:	R_TRIG := (CLK := PTM200StrippedTables[3].Signal);
	
	TurnOnCabinetLights						:	BOOL;
	IgnoreFront								:	BOOL;
	
	CouchLightStepUp: BOOL;
	AllLightsOff: BOOL;
	hmiShutdown: BOOL;
	
	//Dali Diagnostics
	operatingTime							:	FB_DALI253QueryControlGearOperatingTime(Dali.KL6811_Tc3);
END_VAR

//Reset
ReceptionDoorLightControlOnLeave(bOn:= FALSE, bOff:= FALSE,	nAddr:= 24, eAddrType:= 0,stCommandBuffer:= stCommandBuffer);

//Individual Light Control via tLigthTable for direct testing	
FOR i := 0 TO 57 DO
	FBDALIV2Light[i](
			bOn:= tLightTable[i].bOn, 
			bOff:= tLightTable[i].bOff, 
			bToggle:= tLightTable[i].bToggle, 
			nAddr:= i ,
			eAddrType:= 0, 
			nMasterDevAddr:= , 
			tCycleActualLevelMasterDev:= , 
			bLight=> tLightTable[i].LigthStatus, 
			bBusy=> , 
			bError=> , 
			nErrorId=> , 
			stCommandBuffer:= stCommandBuffer);
END_FOR

Update := Update + 1;

(*FOR i := 0 TO 57 DO
	FBDALIV2QueryLightState[i](	
						bStart := update.0,
						nAddr := i,	
						eAddrType := 0,
						bLampPowerOn => tLightTable[i].LigthStatus,
						stCommandBuffer:= stCommandBuffer);
END_FOR	*)

	//force vars
	IF TurnAllOn THEN
	TurnAllOn := FALSE;
	
	LightControlGroup0_MiddleRoom		(bOn:= TRUE, bOff:= , nAddr:= 0, eAddrType:= 1,	bLight=> ,stCommandBuffer:= stCommandBuffer);
	LightControlGroup1_OfficeDesks		(bOn:= TRUE, bOff:= , nAddr:= 1, eAddrType:= 1,	bLight=> ,stCommandBuffer:= stCommandBuffer);
	LightControlGroup2_BoardroomBackRow	(bOn:= TRUE, bOff:= , nAddr:= 2, eAddrType:= 1,	bLight=> ,stCommandBuffer:= stCommandBuffer);
	LightControlGroup3_BoardroomFront2	(bOn:= TRUE, bOff:= , nAddr:= 3, eAddrType:= 1,	bLight=> ,stCommandBuffer:= stCommandBuffer);
	LightControlGroup4_OfficePassage	(bOn:= TRUE, bOff:= , nAddr:= 4, eAddrType:= 1,	bLight=> ,stCommandBuffer:= stCommandBuffer);
	LightControlGroup5_SmallBoardRoom	(bOn:= TRUE, bOff:= , nAddr:= 5, eAddrType:= 1,	bLight=> ,stCommandBuffer:= stCommandBuffer);
	LightControlGroup6_MiddleRoomPassage(bOn:= TRUE, bOff:= , nAddr:= 6, eAddrType:= 1,	bLight=> ,stCommandBuffer:= stCommandBuffer);
	LightControlGroup7_TechRoom			(bOn:= TRUE, bOff:= , nAddr:= 7, eAddrType:= 1,	bLight=> ,stCommandBuffer:= stCommandBuffer);
	LightControlGroup8_ServerRoom		(bOn:= TRUE, bOff:= , nAddr:= 8, eAddrType:= 1,	bLight=> ,stCommandBuffer:= stCommandBuffer);
	
	xXplanarScreenPowerOn := TRUE;
	
	TurnAllOffGroup0_MiddleRoom			(bStart:= FALSE , nAddr:= 0, eAddrType:= 1, stCommandBuffer:= stCommandBuffer );
	TurnAllOffGroup1_OfficeDesks		(bStart:= FALSE , nAddr:= 1, eAddrType:= 1, stCommandBuffer:= stCommandBuffer );		
	TurnAllOffGroup2_BoardroomBackRow	(bStart:= FALSE , nAddr:= 2, eAddrType:= 1, stCommandBuffer:= stCommandBuffer );
	TurnAllOffGroup3_BoardroomFront2	(bStart:= FALSE , nAddr:= 3, eAddrType:= 1, stCommandBuffer:= stCommandBuffer );
	TurnAllOffGroup4_OfficePassage		(bStart:= FALSE , nAddr:= 4, eAddrType:= 1, stCommandBuffer:= stCommandBuffer );
	TurnAllOffGroup5_SmallBoardRoom		(bStart:= FALSE , nAddr:= 5, eAddrType:= 1, stCommandBuffer:= stCommandBuffer );
	TurnAllOffGroup6_MiddleRoomPassage	(bStart:= FALSE , nAddr:= 6, eAddrType:= 1, stCommandBuffer:= stCommandBuffer );
	TurnAllOffGroup7_TechRoom			(bStart:= FALSE , nAddr:= 7, eAddrType:= 1, stCommandBuffer:= stCommandBuffer );	
	TurnAllOffGroup8_ServerRoom			(bStart:= FALSE , nAddr:= 8, eAddrType:= 1, stCommandBuffer:= stCommandBuffer );	
		
	ELSIF TurnAllOFF THEN
	TurnAllOFF := FALSE;	
	LightControlGroup0_MiddleRoom		(bOn:= FALSE, bOff:= , nAddr:= 0, eAddrType:= 1,	bLight=> ,stCommandBuffer:= stCommandBuffer);
	LightControlGroup1_OfficeDesks		(bOn:= FALSE, bOff:= , nAddr:= 1, eAddrType:= 1,	bLight=> ,stCommandBuffer:= stCommandBuffer);
	LightControlGroup2_BoardroomBackRow	(bOn:= FALSE, bOff:= , nAddr:= 2, eAddrType:= 1,	bLight=> ,stCommandBuffer:= stCommandBuffer);
	LightControlGroup3_BoardroomFront2	(bOn:= FALSE, bOff:= , nAddr:= 3, eAddrType:= 1,	bLight=> ,stCommandBuffer:= stCommandBuffer);
	LightControlGroup4_OfficePassage	(bOn:= FALSE, bOff:= , nAddr:= 4, eAddrType:= 1,	bLight=> ,stCommandBuffer:= stCommandBuffer);
	LightControlGroup5_SmallBoardRoom	(bOn:= FALSE, bOff:= , nAddr:= 5, eAddrType:= 1,	bLight=> ,stCommandBuffer:= stCommandBuffer);
	LightControlGroup6_MiddleRoomPassage(bOn:= FALSE, bOff:= , nAddr:= 6, eAddrType:= 1,	bLight=> ,stCommandBuffer:= stCommandBuffer);
	LightControlGroup7_TechRoom			(bOn:= FALSE, bOff:= , nAddr:= 7, eAddrType:= 1,	bLight=> ,stCommandBuffer:= stCommandBuffer);
	LightControlGroup8_ServerRoom		(bOn:= FALSE, bOff:= , nAddr:= 8, eAddrType:= 1,	bLight=> ,stCommandBuffer:= stCommandBuffer);
	
	xXplanarScreenPowerOff := TRUE;
	
	TurnAllOffGroup0_MiddleRoom			(bStart:= TRUE , nAddr:= 0, eAddrType:= 1, stCommandBuffer:= stCommandBuffer );
	TurnAllOffGroup1_OfficeDesks		(bStart:= TRUE , nAddr:= 1, eAddrType:= 1, stCommandBuffer:= stCommandBuffer );		
	TurnAllOffGroup2_BoardroomBackRow	(bStart:= TRUE , nAddr:= 2, eAddrType:= 1, stCommandBuffer:= stCommandBuffer );
	TurnAllOffGroup3_BoardroomFront2	(bStart:= TRUE , nAddr:= 3, eAddrType:= 1, stCommandBuffer:= stCommandBuffer );
	TurnAllOffGroup4_OfficePassage		(bStart:= TRUE , nAddr:= 4, eAddrType:= 1, stCommandBuffer:= stCommandBuffer );
	TurnAllOffGroup5_SmallBoardRoom		(bStart:= TRUE , nAddr:= 5, eAddrType:= 1, stCommandBuffer:= stCommandBuffer );
	TurnAllOffGroup6_MiddleRoomPassage	(bStart:= TRUE , nAddr:= 6, eAddrType:= 1, stCommandBuffer:= stCommandBuffer );
	TurnAllOffGroup7_TechRoom			(bStart:= TRUE , nAddr:= 7, eAddrType:= 1, stCommandBuffer:= stCommandBuffer );	
	TurnAllOffGroup8_ServerRoom			(bStart:= TRUE , nAddr:= 8, eAddrType:= 1, stCommandBuffer:= stCommandBuffer );		
	
	END_IF

IF Bypass THEN
	RETURN;
END_IF

//Set Min or Max for individual lamp ******************************************
	SetMaxLevel(bStart:= xExecuteSetMax, nAddr:= DaliAddrress, eAddrType:= 0, nMaxLevel:= MaxSetting, stCommandBuffer:= stCommandBuffer);

	SetMinLevel(bStart:= xExecuteSetMin, nAddr:= DaliAddrress, eAddrType:= 0, nMinLevel:= MinSetting, stCommandBuffer:= stCommandBuffer);
//******************************************************************************

//Force Lights off after this time*****************************************************************************
GoHomeHold();
ClearRoomTimer();
trigbAssumeBuildingEmpty(CLK := Dali.bAssumeBuildingEmpty);

IF bNoOccupancyFlag THEN
	ResetOthers := FALSE;
	bNoOccupancyFlag := FALSE;
END_IF

IF trigbAssumeBuildingEmpty.Q THEN
	ResetOthers := TRUE;
	TurnAllOffGroup0_MiddleRoom			(bStart:= TRUE , nAddr:= 0, eAddrType:= 1, stCommandBuffer:= stCommandBuffer );
	TurnAllOffGroup1_OfficeDesks		(bStart:= TRUE , nAddr:= 1, eAddrType:= 1, stCommandBuffer:= stCommandBuffer );		
	TurnAllOffGroup2_BoardroomBackRow	(bStart:= TRUE , nAddr:= 2, eAddrType:= 1, stCommandBuffer:= stCommandBuffer );
	TurnAllOffGroup3_BoardroomFront2	(bStart:= TRUE , nAddr:= 3, eAddrType:= 1, stCommandBuffer:= stCommandBuffer );
	TurnAllOffGroup4_OfficePassage		(bStart:= TRUE , nAddr:= 4, eAddrType:= 1, stCommandBuffer:= stCommandBuffer );
	TurnAllOffGroup5_SmallBoardRoom		(bStart:= TRUE , nAddr:= 5, eAddrType:= 1, stCommandBuffer:= stCommandBuffer );
	TurnAllOffGroup6_MiddleRoomPassage	(bStart:= TRUE , nAddr:= 6, eAddrType:= 1, stCommandBuffer:= stCommandBuffer );
	TurnAllOffGroup7_TechRoom			(bStart:= TRUE , nAddr:= 7, eAddrType:= 1, stCommandBuffer:= stCommandBuffer );	
	TurnAllOffGroup8_ServerRoom			(bStart:= TRUE , nAddr:= 8, eAddrType:= 1, stCommandBuffer:= stCommandBuffer );	
	
	xXplanarScreenPowerOff := TRUE;
	
	DeskAreaTriggerOn 			:= FALSE;
	DeskAreaTriggerOff 			:= FALSE;
	SmallBoardRoomTriggerOn		:= FALSE;
	WorkshopPassageTriggerOn 	:= FALSE;
	WorkshopPassageTriggerOff 	:= FALSE;
	OfficePassageTime.IN		:= FALSE;
	WorkshopPassageTime.IN		:= FALSE;
	
	bNoOccupancyFlag := TRUE;
	
END_IF



IF PTM200StrippedTables[5].Signal OR hmiShutdown THEN  // hold in to turn off all before going home
	
	IF  EnOcean.AllWindowsClosed  THEN
		//hmiShutdown := FALSE;
		GoHomeHold.IN := TRUE;	
		GoHomeHold.PT := T#2S;	
			IF GoHomeHold.Q THEN
				GoHomeHold.IN := FALSE;	
				GoHomeHoldActivated := TRUE;
				AllLightsOff := TRUE;
				hmiShutdown := FALSE;
			END_IF	
		xSleepMode := TRUE;		
		
	ELSE
		
		AWindowIsOpenLightTrigger := TRUE;
			
	END_IF		
		
END_IF

IF hmiShutdown THEN  // hold in to turn off all before going home
	
	IF  EnOcean.AllWindowsClosed  THEN
		GoHomeHoldActivated := TRUE;
		AllLightsOff := TRUE;
		hmiShutdown := FALSE;
		xSleepMode := TRUE;		
		
	ELSE
		
		AWindowIsOpenLightTrigger := TRUE;
			
	END_IF		
		
END_IF

IF NOT PTM200StrippedTables[5].Signal AND NOT GoHomeHoldActivated THEN
	GoHomeHold.IN := FALSE;
	TurnAllOffGroup0_MiddleRoom			(bStart:= FALSE , nAddr:= 0, eAddrType:= 1, stCommandBuffer:= stCommandBuffer );
	TurnAllOffGroup1_OfficeDesks		(bStart:= FALSE , nAddr:= 1, eAddrType:= 1, stCommandBuffer:= stCommandBuffer );		
	TurnAllOffGroup2_BoardroomBackRow	(bStart:= FALSE , nAddr:= 2, eAddrType:= 1, stCommandBuffer:= stCommandBuffer );
	TurnAllOffGroup3_BoardroomFront2	(bStart:= FALSE , nAddr:= 3, eAddrType:= 1, stCommandBuffer:= stCommandBuffer );
	TurnAllOffGroup4_OfficePassage		(bStart:= FALSE , nAddr:= 4, eAddrType:= 1, stCommandBuffer:= stCommandBuffer );
	TurnAllOffGroup5_SmallBoardRoom		(bStart:= FALSE , nAddr:= 5, eAddrType:= 1, stCommandBuffer:= stCommandBuffer );
	TurnAllOffGroup6_MiddleRoomPassage	(bStart:= FALSE , nAddr:= 6, eAddrType:= 1, stCommandBuffer:= stCommandBuffer );
	TurnAllOffGroup7_TechRoom			(bStart:= FALSE , nAddr:= 7, eAddrType:= 1, stCommandBuffer:= stCommandBuffer );	
	TurnAllOffGroup8_ServerRoom			(bStart:= FALSE , nAddr:= 8, eAddrType:= 1, stCommandBuffer:= stCommandBuffer );

END_IF

IF GoHomeHoldActivated THEN // Go home swicth has been held
	IgnoreFront := TRUE;
	IgnoreFronttime.IN := IgnoreFront;
	ResetOthers := TRUE;
	
	TurnAllOffGroup0_MiddleRoom			(bStart:= TRUE , nAddr:= 0, eAddrType:= 1, stCommandBuffer:= stCommandBuffer );
	TurnAllOffGroup1_OfficeDesks		(bStart:= TRUE , nAddr:= 1, eAddrType:= 1, stCommandBuffer:= stCommandBuffer );		
	TurnAllOffGroup2_BoardroomBackRow	(bStart:= TRUE , nAddr:= 2, eAddrType:= 1, stCommandBuffer:= stCommandBuffer );
	TurnAllOffGroup3_BoardroomFront2	(bStart:= TRUE , nAddr:= 3, eAddrType:= 1, stCommandBuffer:= stCommandBuffer );
	TurnAllOffGroup4_OfficePassage		(bStart:= TRUE , nAddr:= 4, eAddrType:= 1, stCommandBuffer:= stCommandBuffer );
	TurnAllOffGroup5_SmallBoardRoom		(bStart:= TRUE , nAddr:= 5, eAddrType:= 1, stCommandBuffer:= stCommandBuffer );
	TurnAllOffGroup6_MiddleRoomPassage	(bStart:= TRUE , nAddr:= 6, eAddrType:= 1, stCommandBuffer:= stCommandBuffer );
	TurnAllOffGroup7_TechRoom			(bStart:= TRUE , nAddr:= 7, eAddrType:= 1, stCommandBuffer:= stCommandBuffer );	
	TurnAllOffGroup8_ServerRoom			(bStart:= TRUE , nAddr:= 8, eAddrType:= 1, stCommandBuffer:= stCommandBuffer );	
	
	xXplanarScreenPowerOff := TRUE;

	DeskAreaTriggerOn 			:= FALSE;
	DeskAreaTriggerOff 			:= FALSE;
	SmallBoardRoomTriggerOn		:= FALSE;
	WorkshopPassageTriggerOn 	:= FALSE;
	WorkshopPassageTriggerOff 	:= FALSE;
	OfficePassageTime.IN		:= FALSE;
	WorkshopPassageTime.IN		:= FALSE;
		
	ClearRoomTimer.IN := TRUE;
	ClearRoomTimer.pt := T#100S;
	
	GoHomeHoldActivated := FALSE;
	
	//DMX off
	TurnOnCabinetLights	:= FALSE;
	
END_IF


IgnoreFronttime.pt := T#1S;
IgnoreFronttime();

IF IgnoreFronttime.Q THEN
	IgnoreFronttime.IN := FALSE;
	IgnoreFronttime();
	ReceptionDoorLightControlOnLeave(bOn:= TRUE, bOff:= FALSE,	nAddr:= 24, eAddrType:= 0,stCommandBuffer:= stCommandBuffer);
END_IF

IF ClearRoomTimer.Q THEN
	IgnoreFront := FALSE;
	IgnoreFronttime.IN := FALSE;
	ClearRoomTimer.IN := FALSE;
	ResetOthers := FALSE;
	ReceptionDoorLightControlOnLeave(bOn:= FALSE, bOff:= TRUE,	nAddr:= 24, eAddrType:= 0,stCommandBuffer:= stCommandBuffer);
END_IF


MainEntTimer(IN:= , PT:= T#3600S, Q=> , ET=> );  
OfficeTimer(IN:= , PT:= T#3600S, Q=> , ET=> );  
ReceptionDoorTime(); 
OfficePassageTime();
WorkshopPassageTime();
DeskAreaTime();
BoardRoomTime();

			
//Reception Area**********************************************************
ReceptionDoor_LightControl();
ReceptionPassage_LightControl();



//Dimm Staff Office***************************************************************************
	FBDALIV2Dimmer1SwitchStaff(
	bSwitchDimm:= , 
	bOn:= PTM200StrippedTables[7].Signal, 
	bOff:= PTM200StrippedTables[5].Signal, 
	bSetDimmValue:= , 
	nDimmValue:= , 
	tSwitchOverTime:= , 
	tCycleDelay:= , 
	bMemoryModeOn:= , 
	nOnValueWithoutMemoryMode:= , 
	nAddr:= 1, 
	eAddrType:= 1, 
	nMasterDevAddr:= , 
	nMinLevelMasterDev:= , 
	nMaxLevelMasterDev:= , 
	tCycleActualLevelMasterDev:= , 
	nActualLevelMasterDev=> , 
	bBusy=> , 
	bError=> , 
	nErrorId=> , 
	stCommandBuffer:= stCommandBuffer );

	IF PTM200StrippedTables[6].Signal AND FBDALIV2Dimmer1SwitchStaff.nDimmValue < 254  THEN
		FBDALIV2Dimmer1SwitchStaff.nDimmValue := FBDALIV2Dimmer1SwitchStaff.nDimmValue + 1;
	END_IF		
	
	IF PTM200StrippedTables[4].Signal AND FBDALIV2Dimmer1SwitchStaff.nDimmValue > 0  THEN
		FBDALIV2Dimmer1SwitchStaff.nDimmValue := FBDALIV2Dimmer1SwitchStaff.nDimmValue - 1;
	END_IF	

//Office Light Control***********************************************************************

	//Desk area light control 
	OfficeLightControl(
		bEnable:= TRUE, 
		bOn:= DeskAreaTriggerOn (*PTM200StrippedTables[7].Signal*), 
		bOff:= DeskAreaTriggerOff (*PTM200StrippedTables[5].Signal*), 
		bToggle:= , 
		nSetpointValue:= OfficeLightLevelSetpoint, 
		nActualValue:= Dali.StaffroomPIR_2_LuxLevel, 
		nHysteresis:= 50, 
		nMaxLevel:= 245, 					//250
		nMinLevel:= 10, 
		nStepSize:= 1, 
		tDeadTime:= T#2S, 
		nOptions:= , 
		nDeviation=> , 
		bControllerIsActive=> , 
		bBusy=> , 
		bError=> , 
		nErrorId=> , 
		nLightLevel:= OfficeLightLevel );
		
		FBFadeOffice(
			nDimmValue:= UINT_TO_BYTE(OfficeLightLevel), 
			nAddr:= 1, 
			eAddrType:= 1, 
			stCommandBuffer:= stCommandBuffer);
			
	/////////////////////////// Desk area Occupancy handle //////////////////////////
	IF 	Dali.StaffroomPIR_2_Occupancy  THEN
		DeskAreaTriggerOn 		:= TRUE;
		DeskAreaTriggerOff		:= FALSE;
		DeskAreaTime.IN			:= FALSE;
	END_IF
	
	IF NOT Dali.StaffroomPIR_2_Occupancy THEN
		DeskAreaTime.IN			:= TRUE;
		DeskAreaTime.PT			:= T#1H;	
	END_IF
	
	IF DeskAreaTime.Q OR ResetOthers THEN
		DeskAreaTriggerOn 		:= FALSE;
		DeskAreaTriggerOff		:= TRUE;
	END_IF
	////////////////////////////////////////////////////////////////////////////////////			
		
	//Workshop and server room light control***************************************************************
		LightControlGroup7_TechRoom(
							bOn:= WorkshopPassageTriggerOn, 
							bOff:= WorkshopPassageTriggerOff, 
							nAddr:= 7, 
							eAddrType:= 1, 
							bLight=> , 
							stCommandBuffer:= stCommandBuffer );	
							
		LightControlGroup8_ServerRoom(
							bOn:= WorkshopPassageTriggerOn, 
							bOff:= WorkshopPassageTriggerOff, 
							nAddr:= 8, 
							eAddrType:= 1, 
							bLight=> , 
							stCommandBuffer:= stCommandBuffer );
			
	/////////////////////////// Workshop Passage Occupancy handle //////////////////////////
	IF 	Dali.StaffroomPIR_1_Occupancy  THEN
		WorkshopPassageTriggerOn 		:= TRUE;
		WorkshopPassageTriggerOff		:= FALSE;
		WorkshopPassageTime.IN			:= FALSE;
	END_IF
	
	IF  NOT Dali.StaffroomPIR_1_Occupancy THEN
		WorkshopPassageTime.IN			:= TRUE;
		WorkshopPassageTime.PT			:= T#1H;	
	END_IF
	
	IF WorkshopPassageTime.Q OR ResetOthers THEN

		WorkshopPassageTriggerOn 		:= FALSE;
		WorkshopPassageTriggerOff		:= TRUE;
	END_IF
	////////////////////////////////////////////////////////////////////////////////////		
			
	
//Office passge light control**********************************************************
		OfficePassageLightControl(
			bOn:= OfficePassageTriggerOn, 
			bOff:= OfficePassageTriggerOFF,
			nAddr:= 4, 
			eAddrType:= 1, 
			nMasterDevAddr:= , 
			tCycleActualLevelMasterDev:= , 
			stCommandBuffer:= stCommandBuffer);	
			
				

//Small Board Room Group 5**********************************************************
LightControlGroup5_SmallBoardRoom(
			bOn:= SmallBoardRoomTriggerOn, 
			bOff:= SmallBoardRoomTriggerOFF,
			nAddr:= 5, 
			eAddrType:= eDALIV2AddrTypeGroup, 
			stCommandBuffer:= stCommandBuffer);		
			
//RecallMinLevelGroup5_SmallBoardRoom(
//			bStart:= SmallBoardRoomTriggerOn,
//			nAddr:= 5, 
//			eAddrType:= eDALIV2AddrTypeGroup, 
//			stCommandBuffer:= stCommandBuffer );
//SmallBoardRoomOff(
//			bStart:= TRUE, 
//			nAddr:= 55, 
//			eAddrType:= eDALIV2AddrTypeShort,  
//			stCommandBuffer:= stCommandBuffer);
//*******************************************************************************
		
	
/////////////////////////// Office Passage Occupancy handle //////////////////////////
IF 	Dali.StaffroomPIR_1_Occupancy OR Dali.StaffroomPIR_2_Occupancy  THEN
	OfficePassageTriggerOn 		:= TRUE;
	OfficePassageTriggerOFF		:= FALSE;
	OfficePassageTime.IN		:= FALSE;
END_IF

IF NOT Dali.StaffroomPIR_1_Occupancy AND NOT Dali.StaffroomPIR_2_Occupancy THEN
	OfficePassageTime.IN		:= TRUE;
	OfficePassageTime.PT		:= T#1H;	
END_IF

IF OfficePassageTime.Q OR ResetOthers THEN

	OfficePassageTriggerOn 		:= FALSE;
	OfficePassageTriggerOFF		:= TRUE;
END_IF
////////////////////////////////////////////////////////////////////////////////////

bLightADS := PTM200StrippedTables[3].Signal;
bLightsADSOff := 	PTM200StrippedTables[1].Signal;
bLightsADSOff := 	PTM200StrippedTables[0].Signal;

//All Board room on********************************************************************
BoardRoom_LightControl();	
//Board table spots****************************************************

	FOR i := 10 TO 11 DO
	FBDALIV2Light[i](
		bOn:= PTM200StrippedTables[3].Signal, 
		bOff:= PTM200StrippedTables[0].Signal, 
		bToggle:= , 
		nAddr:= i, 
		eAddrType:= 0, 
		nMasterDevAddr:= , 
		tCycleActualLevelMasterDev:= , 
		bLight=> , 
		stCommandBuffer:= stCommandBuffer );
	END_FOR	
	
	FOR i := 10 TO 11 DO
	FBDALIV2Light[i](
		bOn:= PTM200StrippedTables[3].Signal, 
		bOff:= PTM200StrippedTables[0].Signal, 
		bToggle:= , 
		nAddr:= i, 
		eAddrType:= 0, 
		nMasterDevAddr:= , 
		tCycleActualLevelMasterDev:= , 
		bLight=> , 
		stCommandBuffer:= stCommandBuffer );
	END_FOR	

				

	/////////////////////////// Office Passage Occupancy handle //////////////////////////
	IF 	Dali.CommunalAreaPIR_2_Occupancy AND NOT ReceptionTableKitchLoungeLightControl.bLight THEN
		ReceptionTableKitchLoungeTriggerOn 		:= TRUE;
		ReceptionTableKitchLoungeTriggerOFF		:= FALSE;
		ReceptionTableKitchLoungeTime.IN		:= FALSE;
	END_IF
	
	IF NOT Dali.CommunalAreaPIR_2_Occupancy  THEN
		ReceptionTableKitchLoungeTime.IN		:= TRUE;
		ReceptionTableKitchLoungeTime.PT		:= T#1H;	
	END_IF
	
	IF ReceptionTableKitchLoungeTime.Q OR ResetOthers THEN

		ReceptionTableKitchLoungeTriggerOn 		:= FALSE;
		ReceptionTableKitchLoungeTriggerOFF		:= TRUE;
	END_IF
	
	//Reception Kitch.lounge.table light control**********************************************************
		ReceptionTableKitchLoungeLightControl(
			bOn:= ReceptionTableKitchLoungeTriggerOn, 
			bOff:= ReceptionTableKitchLoungeTriggerOFF,
			nAddr:= 0, 
			eAddrType:= 1, 
			nMasterDevAddr:= , 
			bLight => ,
			tCycleActualLevelMasterDev:= , 
			stCommandBuffer:= stCommandBuffer);	
			
		(*RecallMinLevelGroup5_SmallBoardRoom(
			bStart:= ReceptionTableKitchLoungeTriggerOn, 
			nAddr:= 5, 
			eAddrType:= eDALIV2AddrTypeGroup, 
			stCommandBuffer:= stCommandBuffer );*)
			
		(*RecallMinLevelCouchLight(
			bStart:= ReceptionTableKitchLoungeTriggerOn, 
			nAddr:= 57, 
			eAddrType:= eDALIV2AddrTypeShort    , 
			stCommandBuffer:= stCommandBuffer );*)
		
		RecallStepUPCouchLight(
			bStart:= CouchLightStepUp, 
			nAddr:= 57, 
			eAddrType:= eDALIV2AddrTypeShort, 
			stCommandBuffer:= stCommandBuffer);
	
	
	IF ReceptionTableKitchLoungeTriggerOn THEN
		ReceptionTableKitchLoungeTriggerOn := FALSE;
		xXplanarScreenPowerOn := TRUE;	
	END_IF 		
	
	IF ReceptionTableKitchLoungeTriggerOff THEN
		ReceptionTableKitchLoungeTriggerOff := FALSE;
		
	END_IF 		
	
	////////////////////////////////////////////////////////////////////////////////////
	operatingTime(
		bError=> , 
		ipResultMessage=> , 
		bStart:= , 
		nAddress:= 5, 
		eAddressType:= E_DALIAddressType.Short, 
		eCommandPriority:= E_DALICommandPriority.MiddleLow, 
		bBusy=> , 
		nControlGearOperatingTime=> );

ACTION BoardRoom_LightControl:
/////////////////////////// Boardroom area Occupancy handle //////////////////////////
IF 	Dali.BoardroomPIR_1_Occupancy OR Dali.BoardroomPIR_2_Occupancy THEN
	BoardRoomTriggerOn 		:= TRUE;
	BoardRoomTriggerOff		:= FALSE;
	BoardRoomTime.IN		:= FALSE;
END_IF

IF (NOT Dali.BoardroomPIR_2_Occupancy) OR (NOT Dali.BoardroomPIR_1_Occupancy) OR rt_BoardRoom_Lights_ProjectorMode.Q OR rt_BoardRoom_Lights_ShowroomMode.Q THEN
	BoardRoomTime.IN			:= TRUE;
	BoardRoomTime.PT			:= T#0.4H;	
END_IF

IF BoardRoomTime.Q OR ResetOthers OR rt_BoardRoom_Lights_Switch0.Q OR rt_BoardRoom_Lights_Switch1.Q THEN	//OR PTM200StrippedTables[1].Signal or PTM200StrippedTables[0].Signal 
	BoardRoomTriggerOn 		:= FALSE;
	BoardRoomTriggerOff		:= TRUE;
END_IF

//Showroom Board room on*********************************************

rt_BoardRoom_Lights_ShowroomMode(CLK := xBoardRoom_Lights_ShowroomMode);

IF  rt_BoardRoom_Lights_ShowroomMode.Q THEN
	xBoardRoom_Lights_ShowroomMode := FALSE;
	BoardRoomTriggerOn		:= TRUE;
	BoardRoomTriggerOff		:= FALSE;
	BoardRoomTime.IN		:= FALSE;
END_IF

FBDALIV2Dimmer1SwitchBoarda(
	bSwitchDimm:= , 
	bOn:= PTM200StrippedTables[2].Signal OR BoardRoomTriggerOn, 
	bOff:= PTM200StrippedTables[0].Signal OR BoardRoomTriggerOff OR rt_BoardRoom_Lights_ProjectorMode.Q , 
	nAddr:= 3, 
	eAddrType:= 1, 
	stCommandBuffer:= stCommandBuffer); 

FBDALIV2Dimmer1SwitchBoardb(
	bSwitchDimm:= , 
	bOn:= PTM200StrippedTables[2].Signal OR BoardRoomTriggerOn, 
	bOff:= PTM200StrippedTables[0].Signal OR BoardRoomTriggerOff, 
	nAddr:= 2, 
	eAddrType:= 1, 
	stCommandBuffer:= stCommandBuffer );	



//Projector Board room on*********************************************

rt_BoardRoom_Lights_ProjectorMode(CLK := xBoardRoom_Lights_ProjectorMode);

IF  rt_BoardRoom_Lights_ProjectorMode.Q THEN
	xBoardRoom_Lights_ProjectorMode := FALSE;
	BoardRoomTriggerOff		:= FALSE;
	BoardRoomTime.IN		:= FALSE;
END_IF

FBDALIV2Dimmer1SwitchBoardc(
	bSwitchDimm:= , 
	bOn:= rt_BoardRoom_Lights_ShowroomMode.Q, 
	bOff:= PTM200StrippedTables[1].Signal OR rt_BoardRoom_Lights_ProjectorMode.Q OR BoardRoomTriggerOff, //Bottom Left Switch
	nAddr:= 3, 
	eAddrType:= 1, 
	stCommandBuffer:= stCommandBuffer );

FBDALIV2Dimmer1SwitchBoardd(
	bSwitchDimm:= , 
	bOn:= PTM200StrippedTables[3].Signal OR rt_BoardRoom_Lights_ProjectorMode.Q, //Bottom Right Switch
	bOff:= PTM200StrippedTables[1].Signal or BoardRoomTriggerOff,  //Bottom Left Switch
	nAddr:= 2, 
	eAddrType:= 1, 
	stCommandBuffer:= stCommandBuffer );
END_ACTION

ACTION ReceptionDoor_LightControl:
//Reception Door light control**********************************************************
IF NOT IgnoreFront THEN

		ReceptionDoorLightControl(
			bOn:= ReceptionDoorTriggerOn, 
			bOff:= , //ReceptionDoorTriggerOFF
			nAddr:= 24, 
			eAddrType:= 0, 
			nMasterDevAddr:= , 
			tCycleActualLevelMasterDev:= , 
			stCommandBuffer:= stCommandBuffer);	

	/////////////////////////// Reception Door  Occupancy handle //////////////////////////
	IF 	Dali.CommunalAreaPIR_1_Occupancy  THEN
		
		ReceptionDoorTriggerOn 		:= TRUE;
		ReceptionDoorTriggerOFF		:= FALSE;
		ReceptionDoorTime.IN		:= FALSE;
		TurnOnCabinetLights			:= TRUE;
		AllLightsOff				:= FALSE;
	END_IF
	
	IF NOT Dali.CommunalAreaPIR_1_Occupancy  THEN
		ReceptionDoorTime.IN		:= TRUE;
		ReceptionDoorTime.PT		:= T#3600S;	
	END_IF
	
	IF ReceptionDoorTime.Q OR ResetOthers THEN
		TurnOnCabinetLights := FALSE;
		ReceptionDoorTriggerOn 		:= FALSE;
		ReceptionDoorTriggerOFF		:= TRUE;
	END_IF
	//***************************************************************************************

	
END_IF
END_ACTION

ACTION ReceptionPassage_LightControl:
//Reception Passage light control**********************************************************
		ReceptionPassageLightControl(
			bOn:= ReceptionPassageTriggerOn, 
			bOff:= ReceptionPassageTriggerOFF,
			nAddr:= 6, 
			eAddrType:= 1, 
			nMasterDevAddr:= , 
			tCycleActualLevelMasterDev:= , 
			stCommandBuffer:= stCommandBuffer);	

	/////////////////////////// Reception Passage  Occupancy handle //////////////////////////
	IF 	Dali.StaffroomPIR_1_Occupancy OR Dali.StaffroomPIR_2_Occupancy OR Dali.CommunalAreaPIR_2_Occupancy THEN
		SmallBoardRoomTriggerOn				:= TRUE;		//to be changed
		ReceptionPassageTriggerOn 			:= TRUE;
		ReceptionPassageTriggerOFF			:= FALSE;
		ReceptionPassageTime.IN				:= FALSE;
		SmallBoardRoomTime.IN				:= FALSE;		//to be changed
	END_IF
	
	IF NOT Dali.StaffroomPIR_1_Occupancy AND NOT Dali.StaffroomPIR_2_Occupancy AND NOT Dali.CommunalAreaPIR_2_Occupancy THEN
		ReceptionPassageTime.IN				:= TRUE;
		SmallBoardRoomTime.IN				:= TRUE;
		ReceptionPassageTime.PT				:= T#3600S;
		SmallBoardRoomTime.PT				:= T#3600S;	
	END_IF
	
	IF ReceptionPassageTime.Q OR ResetOthers THEN
		SmallBoardRoomTriggerOn				:= FALSE;
		ReceptionPassageTriggerOn 			:= FALSE;
		ReceptionPassageTriggerOFF			:= TRUE;
		SmallBoardRoomTriggerOFF			:= True;
	END_IF
	//***************************************************************************************
END_ACTION

END_PROGRAM

// ---- HMI/FileHandle.TcPOU
PROGRAM FileHandle
VAR
	///File Handle Blocks from Tc2_System.lib
	fbOpenFile: FB_FileOpen;
	fbWriteFile: FB_FilePuts;
	fbReadFile: FB_FileRead;
	fbCloseFile: FB_FileClose;
	///Case Variables
	nFileCaseIndex: INT;
	nSignOutCase: INT;
	nWriteTableCase: INT;
	///DateTime
	fbGetTime: NT_GetTime;
	///Triggers and GeneralVars
	rtSignInTrig: R_TRIG;
	rtSignOut: R_TRIG;
	rtChangeMade: R_TRIG;
	i: INT;
	y: INT;
	///File Variables
	sFileName: STRING;
	sLine: STRING(255);
	Init: BOOL;
	DateChange: STRING;
	MonthEnd: BOOL;
END_VAR

//Get and format system time
GetSystemTime();

//Init IF
IF NOT Init THEN
	Init := TRUE;
	DateChange := STDateTimeStrings.sDay;
END_IF

IF DateChange <> STDateTimeStrings.sDay THEN //See if date has changed to save table and clear it for new month
	DateChange :=  STDateTimeStrings.sDay;
	CurrentMonthSignInTable := BlankCurrentMonthSignInTable;
	ComboBoxCurrentMonthSignInTable := BlankComboBoxCurrentMonthSignInTable;
	rtChangeMade.CLK := TRUE;
END_IF

//Hide sign in button
IF sVisuName = '' OR sVisuCompany = '' OR sVisuPersonVisiting = '' THEN
	xVisuHideSignInButton := TRUE;
ELSE	
	xVisuHideSignInButton := FALSE;
END_IF

//Sign in clicked?	
rtSignInTrig(CLK:= xVisuSignInButton);

IF rtSignInTrig.Q THEN
	xVisuSignInButton := FALSE;
	rtChangeMade.CLK := TRUE;
	nWriteTableCase := 10;
END_IF

//SignOutWith
	rtSignOut(CLK:= xVisuSignOutButton);
	
	IF rtSignOut.Q AND CurrentMonthSignInTable[nVisuTableRowSelection].Name <> '' THEN
		xVisuSignOutButton := FALSE;
		CurrentMonthSignInTable[nVisuTableRowSelection].sTimeOut := sTime;
		//CurrentMonthSignInTable[nVisuTableRowSelection].Email := sVisuEmailAddress;
		//sVisuEmailAddress := '';
		//CurrentMonthSignInTable[nVisuTableRowSelection].PCControl := xVisuYesPCControl;
		//xVisuYesPCControl := FALSE;
		CurrentMonthSignInTable[nVisuTableRowSelection].SignOut := TRUE; 
		rtChangeMade.CLK := TRUE;
		nSignOutCase := 10;
	END_IF

//Change Made to table, trigger file write
rtChangeMade();

IF rtChangeMade.Q THEN
	nFileCaseIndex := 10;
	rtChangeMade.CLK := FALSE;
END_IF

	//Move customer info to table case
	CASE nWriteTableCase OF
		
	0:	//IDLE	

	10:	//Write customer details to table and file
		xVisuSignInButton := FALSE;
		FOR  i := 0 TO nMaxTableLength DO
			IF CurrentMonthSignInTable[i].Name = '' THEN
				
			ComboBoxCurrentMonthSignInTable[i]			:= sVisuName;
						
			CurrentMonthSignInTable[i].Name 				:= sVisuName; 
			CurrentMonthSignInTable[i].Company 			:= sVisuCompany; 
			CurrentMonthSignInTable[i].PersonVisiting 	:= sVisuPersonVisiting; 
			CurrentMonthSignInTable[i].Reason		 	:= sVisuReason; 
			CurrentMonthSignInTable[i].VehicleReg 		:= sVisuVehicleReg; 
			CurrentMonthSignInTable[i].sDate		 		:= sDate; 
			CurrentMonthSignInTable[i].sTimeIn		 	:= sTime; 
			CurrentMonthSignInTable[i].PCControl		 	:= xVisuYesPCControl;
			CurrentMonthSignInTable[i].Email			 	:= sVisuEmailAddress; 
	
			
			EXIT;		
			END_IF
		END_FOR
		
		nWriteTableCase := 20;
		
	20:		
			sVisuName := '';
			sVisuCompany := '';
			sVisuPersonVisiting := ''; 
			sVisuReason := ''; 
			sVisuVehicleReg := ''; 
			sDate := ''; 
			sTime := ''; 
			xVisuYesPCControl := FALSE;
			sVisuEmailAddress := ''; 
		
		nWriteTableCase := 0;	

				
	END_CASE
	
	
// Write changes to file
	
CASE nFileCaseIndex OF
	
0:	//Idle, waiting for a change to be made
	
10:	fbOpenFile.sPathName := '\Hard Disk\SignIn\';
	fbOpenFile.sPathName :=  CONCAT(fbOpenFile.sPathName , sFileName );
	fbOpenFile.sPathName :=  CONCAT(fbOpenFile.sPathName , '.csv' );

	fbOpenFile(sNetId:= , nMode:= FOPEN_MODEWRITE, bExecute:= TRUE, tTimeout:= T#2S);
	
	nFileCaseIndex := 20;
	
20:	fbOpenFile(bExecute := FALSE);	
	IF NOT fbOpenFile.bBusy THEN
		
		IF CurrentMonthSignInTable[y].Name <> '' THEN
			BuildFileString();			
			fbWriteFile(hFile := fbOpenFile.hFile , 
			sLine:= sLine, 
			bExecute:= TRUE, 
			tTimeout:= T#2S );	
			nFileCaseIndex := 30;
		ELSE
			nFileCaseIndex := 30;	
		END_IF
	
	END_IF
	
30:	fbWriteFile();
	IF NOT fbWriteFile.bBusy THEN
		fbWriteFile(bExecute := FALSE);
		y := y + 1;
		
		IF CurrentMonthSignInTable[y].Name <> '' THEN
			nFileCaseIndex := 20;	
		ELSE
			nFileCaseIndex := 40;	
		END_IF
		
	END_IF;

40: fbCloseFile(hFile:= fbOpenFile.hFile , 
	bExecute:= TRUE, 
	tTimeout:= T#2S);
	y := 0;
	nFileCaseIndex := 50;	
	
50:	fbCloseFile();
	IF NOT fbCloseFile.bBusy THEN
		fbCloseFile(bExecute := FALSE);
		nFileCaseIndex := 0;
	END_IF

END_CASE

ACTION BuildFileString:

	
	sLine := 	CurrentMonthSignInTable[y].Name ;
	sLine :=	CONCAT(sLine, ',');
	sLine :=	CONCAT(sLine, 	CurrentMonthSignInTable[y].Company);
	sLine :=	CONCAT(sLine, ',');
	sLine :=	CONCAT(sLine, 	CurrentMonthSignInTable[y].PersonVisiting);
	sLine :=	CONCAT(sLine, ',');
	sLine :=	CONCAT(sLine, 	CurrentMonthSignInTable[y].Reason);
	sLine :=	CONCAT(sLine, ',');
	sLine :=	CONCAT(sLine, 	CurrentMonthSignInTable[y].VehicleReg);
	sLine :=	CONCAT(sLine, ',');
	sLine :=	CONCAT(sLine, 	CurrentMonthSignInTable[y].sDate);
	sLine :=	CONCAT(sLine, ',');
	sLine :=	CONCAT(sLine, 	CurrentMonthSignInTable[y].sTimeIn);	
	sLine :=	CONCAT(sLine, ',');
	sLine :=	CONCAT(sLine, 	BOOL_TO_STRING(CurrentMonthSignInTable[y].SignOut));
	sLine :=	CONCAT(sLine, ',');
	sLine :=	CONCAT(sLine, 	CurrentMonthSignInTable[y].sTimeOut);
	sLine :=	CONCAT(sLine, ',');
	sLine :=	CONCAT(sLine, 	BOOL_TO_STRING(CurrentMonthSignInTable[y].PCControl));
	sLine :=	CONCAT(sLine, ',');
	sLine :=	CONCAT(sLine, 	CurrentMonthSignInTable[y].Email	);
	sLine :=	CONCAT(sLine, '$L');
END_ACTION

ACTION GetSystemTime:
fbGetTime(NETID:= , START:= TRUE , TMOUT:= T#2S, BUSY=> , ERR=> , ERRID=> , TIMESTR=> );
fbGetTime(NETID:= , START:= FALSE, TMOUT:= T#2S, BUSY=> , ERR=> , ERRID=> , TIMESTR=> );

STDateTimeStrings.sYear := WORD_TO_STRING(fbGetTime.TIMESTR.wYear);

IF fbGetTime.TIMESTR.wMonth > 9 THEN
STDateTimeStrings.sMonth := WORD_TO_STRING(fbGetTime.TIMESTR.wMonth);
ELSE
STDateTimeStrings.sMonth := '0';
STDateTimeStrings.sMonth := CONCAT(STDateTimeStrings.sMonth,WORD_TO_STRING(fbGetTime.TIMESTR.wMonth));
END_IF

IF fbGetTime.TIMESTR.wDay > 9 THEN
STDateTimeStrings.sDay := WORD_TO_STRING(fbGetTime.TIMESTR.wDay);
ELSE
STDateTimeStrings.sDay := '0';
STDateTimeStrings.sDay := CONCAT(STDateTimeStrings.sDay,WORD_TO_STRING(fbGetTime.TIMESTR.wDay));
END_IF

IF fbGetTime.TIMESTR.wHour > 9 THEN
STDateTimeStrings.sHour := WORD_TO_STRING(fbGetTime.TIMESTR.wHour);
ELSE
STDateTimeStrings.sHour := '0';
STDateTimeStrings.sHour := CONCAT(STDateTimeStrings.sHour,WORD_TO_STRING(fbGetTime.TIMESTR.wHour));
END_IF

IF fbGetTime.TIMESTR.wMinute > 9 THEN
STDateTimeStrings.sMinute := WORD_TO_STRING(fbGetTime.TIMESTR.wMinute);
ELSE
STDateTimeStrings.sMinute := '0';
STDateTimeStrings.sMinute := CONCAT(STDateTimeStrings.sMinute,WORD_TO_STRING(fbGetTime.TIMESTR.wMinute));
END_IF

IF fbGetTime.TIMESTR.wSecond > 9 THEN
STDateTimeStrings.sSecond := WORD_TO_STRING(fbGetTime.TIMESTR.wSecond);
ELSE
STDateTimeStrings.sSecond := '0';
STDateTimeStrings.sSecond := CONCAT(STDateTimeStrings.sSecond,WORD_TO_STRING(fbGetTime.TIMESTR.wSecond));
END_IF


sDate :=  STDateTimeStrings.sDay;
sDate := CONCAT(sDate,'/');
sDate := CONCAT(sDate,STDateTimeStrings.sMonth);
sDate := CONCAT(sDate,'/');
sDate := CONCAT(sDate,STDateTimeStrings.sYear);

sTime :=  STDateTimeStrings.sHour;
sTime := CONCAT(sTime,':');
sTime := CONCAT(sTime,STDateTimeStrings.sMinute);
sTime := CONCAT(sTime,':');
sTime := CONCAT(sTime,STDateTimeStrings.sSecond);

sFileName := CONCAT(STDateTimeStrings.sDay , STDateTimeStrings.sMonth);
sFileName := CONCAT(sFileName , STDateTimeStrings.sYear);
END_ACTION

END_PROGRAM

// ---- HMI/TableTennisScoreCounter.TcPOU
PROGRAM TableTennisScoreCounter
VAR

	nPlayerOne			:	INT;
	nPlayerTwo			:	INT;
	nPlayerScoreDiff	:	INT;
	
	sPlayerOne			:	STRING;
	sPlayerTwo			:	STRING;
	
	sPlayerList: ARRAY [0..nMaxTableLength] OF STRING := ['Adam', 'Alan', 'Astrid', 'Jamie', 'Ivo', 'Guest', 'Guest'];
		
	sWinner 			: 	STRING;	
	
	xPlayerOneWins		:	BOOL;	
	xPlayerTwoWins		:	BOOL;	
	
	rtPlayerOne			:	R_TRIG;	
	rtPlayerTwo			:	R_TRIG;
	rtResetOne			:	R_TRIG;
	rtResetTwo			:	R_TRIG;
	
	gameMode5s			:	BOOL;
	
	i: INT;
END_VAR

rtPlayerOne(CLK := PTM200StrippedTables[12].Signal);
rtPlayerTwo(CLK := PTM200StrippedTables[13].Signal);
rtResetOne(CLK := PTM200StrippedTables[14].Signal);
rtResetTwo(CLK := PTM200StrippedTables[15].Signal);



IF rtPlayerOne.Q THEN
	nPlayerOne := nPlayerOne + 1;
END_IF

IF rtPlayerTwo.Q THEN
	nPlayerTwo := nPlayerTwo + 1;
END_IF

IF rtResetOne.Q THEN
	nPlayerOne := 0;
END_IF

IF rtResetTwo.Q THEN
	nPlayerTwo := 0;
END_IF

IF gameMode5s THEN
	Play5s();
ELSE
	Play11s();
END_IF

nPlayerScoreDiff := ABS(nPlayerOne - nPlayerTwo);

IF nPlayerOne >= 11 AND nPlayerOne > nPlayerTwo AND nPlayerScoreDiff >= 2 THEN
	sWinner := CONCAT(sPlayerOne, ' Wins');
	xPlayerOneWins := TRUE;
ELSIF nPlayerTwo >= 11 AND nPlayerTwo > nPlayerOne AND nPlayerScoreDiff >= 2 THEN
	sWinner := CONCAT(sPlayerTwo, ' Wins');
	xPlayerTwoWins := TRUE;
END_IF

